(* IEC 61131-3 sources: elnaProjects/ElpcLogic/PomarKc7Changed/build_USO_ecl/_ (part 3) *)

  IF NOT onInit THEN
           fb_timer480(phaseNumber:=1, delay:=T#480S);
           fb_kran4Open(phaseNumber:=2, act:=_on);
           fb_waitAfterKran4(phaseNumber:=3, delay:=T#10S);
           fb_kran5Close(phaseNumber:=4, act:=_off);
           fb_kran3bOpen(phaseNumber:=5, act:=_on);
           fb_dP_kr1less100(phaseNumber:=6);
           fb_Pvh_vyhMore5(phaseNumber:=7);
           fb_kran1Open(phaseNumber:=8, act:=_on);
           fb_kran2Open(phaseNumber:=9, act:=_on);
           fb_kran3Open(phaseNumber:=10, act:=_on);
           fb_kran3bClose(phaseNumber:=11, act:=_off);
           fb_Err_ALG(phaseNumber:=12);
  onInit:=TRUE;
  END_IF;

  fb_timer480(StrPh:=timer480);
  fb_kran4Open(StrPh:= kran4Open, Im:=Im.kran4);
  fb_waitAfterKran4(StrPh:= waitAfterKran4);
  fb_kran5Close(StrPh:=kran5Close, Im:=Im.kran5);
  fb_kran3bOpen(StrPh:=kran3bOpen, Im:=Im.kran3b);
  fb_dP_kr1less100(StrPh:=dP_kr1less100);
  fb_Pvh_vyhMore5(StrPh:=Pvh_vyhMore5);
  fb_kran1Open(StrPh:=kran1Open, Im:=Im.kran1);
  fb_kran2Open(StrPh:=kran2Open, Im:=Im.kran2);
  fb_kran3Open(StrPh:=kran3Open, Im:=Im.kran3);
  fb_kran3bClose(StrPh:=kran3bClose, Im:=Im.kran3b);
  fb_Err_ALG(StrPh:=Err_ALG);

  StrAlg.CanRun := StrAlg.inCanRun;
  StrAlg.OpcCommandsDisabled := StrAlg.inOpcCommandsDisabled;

  IF StrAlg.isRuning THEN
      (* запуск таймера *)
      IF NOT (kran3bClose.top) THEN
  	    runPhase(timer480);
      END_IF;

      (*если кран1 не открыт - октрыть кран 4*)
      IF	NOT kran1Open.top (*AND IM.kran4._cmdreset.IN = FALSE*)  THEN
  	    runIfNotRunningSO(IM.SingleOutputs.Kr4_open_from_alg);
  	    runPhase(kran4Open);
      END_IF;
      IF	kran4Open.start AND NOT kran4Open.top THEN
  	    IF	IM.kran4.onStatus = _statusDualInput.STATUS_ON THEN
  		    kran4Open.top:=TRUE;
  	    END_IF;
      END_IF;

      (* продувка крана *)
      IF kran4Open.top THEN
          runPhase(waitAfterKran4);
      END_IF;

      (* кран продулся - закрытие кран 5*)
      IF waitAfterKran4.top THEN
  	    runPhase(kran5Close);
      END_IF;

      (* кран 5 закрыт - открытие крана 3б проверка перепада давление*)
      IF	kran5Close.top THEN
  	    runPhase(kran3bOpen);
  	    runPhase(dP_kr1less100);
  	    runPhase(Pvh_vyhMore5);
      END_IF;

      (* проверка давления крана *)
      IF	Pvh_vyhMore5.start AND NOT Pvh_vyhMore5.top THEN
  	    IF	(ai.Pgaza_na_vhode_nagnetatelia.interval >=statusAi.NORMAL) AND (ai.Pgaza_na_vhode_nagnetatelia.value	 >= 4.0) AND
  		    (ai.Pgaza_na_vyhode_nagnetatelia.interval >=statusAi.NORMAL) AND (ai.Pgaza_na_vyhode_nagnetatelia.value	 >= 4.0) THEN
  		        Pvh_vyhMore5.top := TRUE;
      		    runAiProtection(protections.Pgaza_na_vyhode_nagnetatelia);
  	    END_IF;
      END_IF;

      (* проверка открытия крана 3б *)
      IF	kran3bOpen.start AND NOT kran3bOpen.top THEN
  	    IF	IM.kran3b.onStatus=_statusDualInput.STATUS_ON THEN
  		    kran3bOpen.top :=TRUE;
  	    END_IF;
      END_IF;
      IF	kran3bOpen.top AND	kran5Close.top AND dP_kr1less100.top AND Pvh_vyhMore5.top THEN
  	    runPhase(kran1Open);
  	    runPhase(kran2Open);
  	    runPhase(kran3Open);
  	    (*Smazka_1_2:=TRUE; нет такого *)
      END_IF;
      IF	kran1Open.top THEN
  	    resetIfRunningSO(IM.SingleOutputs.Kr4_open_from_alg);
  	    (*ystavki.Block_kr4_alg.setValue (0);что такое уставки*)
      END_IF;

      (* закрытие крана 3бис *)
      IF kran1Open.top AND kran2Open.top AND kran3Open.top THEN
  	    runPhase(kran3bClose);
      END_IF;
      IF 	kran3bClose.top THEN
  	    Err_ALG.error :=FALSE;
  	    resetPhase(timer480);
      ELSIF NOT kran3bClose.top AND timer480.top THEN
  		Err_ALG.error :=TRUE;
      END_IF;
  END_IF;

  _sunpackerCommand(command := StrAlg.inCommand);
  	source := _sunpackerCommand.source;
  	cmd := _sunpackerCommand.cmd;

  IF cmd <> 0 AND lastCmd <> cmd AND (((NOT StrAlg.opcCommandsDisabled) AND source > 0) OR source = 0) then
  	CASE BYTE_TO_INT(cmd) OF
  		(*cmdRun*) 1: 	IF (StrAlg.CanRun) THEN
  					StrAlg.isRuning := TRUE;
  					StrAlg.isEnded := FALSE;
  					StrAlg.hasError := FALSE;
  					(*****************       OnRun       *****************)
                                                    algManager.nMode:=ModeGpa.MODE_PUSK_FIRST_FAZA2;

                                                    (*runPhase(timer120);
                                                    runPhase(timer5);
                                                    runPhase(Shup);
                                                    resetAiProtection(protections.dPmaslo_gaz);
                                                    resetDiProtection(protections.dPmaslo_gaz_less100);*)

  					cmd_for_Status := cmd;
  					source_for_Status := source;
  					command_error_for_Status := 0;
  				ELSE
  					StrAlg.isRuning := FALSE;
  					StrAlg.isEnded := FALSE;
  					StrAlg.hasError := FALSE;

  					cmd_for_Status := 0;
  					source_for_Status := source;
  					command_error_for_Status := cmd;
  				END_IF;
  		(*cmdReset*) 2: 	StrAlg.isRuning := FALSE;
  				StrAlg.isEnded := FALSE;
  				StrAlg.hasError 	:= FALSE;

                                           (*****************       OnReset       *****************)
                                          waitReset(IN:=FALSE);
                                          StrAlg.inCanRun:=FALSE;

                                          (*resetPhase(timer5);
                                          resetPhase(Shup);
                                          resetPhase(timer120);
                                          resetPhase(Net_Chast);
                                          resetPhase(mvOn);
                                          resetPhase(pGNSmore04);
                                          resetPhase(gotov_K_zagruzke);
                                          resetPhase(dPmg_Top);
                                          resetPhase(AutoPNS_Start);*)

                                          StrAlg.inOpcCommandsDisabled:=FALSE;

  				cmd_for_Status := cmd;
  				source_for_Status := source;
  				command_error_for_Status := 0;
  	END_CASE;
  	resetCmdTimer(IN := false);
  	resetCmdTimerPriznak := TRUE;
  END_IF;
  lastCmd := cmd;

  resetCmdTimer(IN := resetCmdTimerPriznak, PT := T#5S);
  IF resetCmdTimer.Q THEN
  	resetCmdTimerPriznak := FALSE;
  	source_for_Status := 0;
  	cmd_for_Status := 0;
  	command_error_for_Status := 0;
  END_IF;

  StrAlg.Start:= timer480.startStatus
              OR kran4Open.startStatus
              OR waitAfterKran4.startStatus
              OR kran5Close.startStatus
              OR kran3bOpen.startStatus
              OR dP_kr1less100.startStatus
              OR Pvh_vyhMore5.startStatus
              OR kran1Open.startStatus
              OR kran2Open.startStatus
              OR kran3Open.startStatus
              OR kran3bClose.startStatus
              OR Err_ALG.startStatus;

  StrAlg.Error := timer480.errorStatus
              OR kran4Open.errorStatus
              OR waitAfterKran4.errorStatus
              OR kran5Close.errorStatus
              OR kran3bOpen.errorStatus
              OR dP_kr1less100.errorStatus
              OR Pvh_vyhMore5.errorStatus
              OR kran1Open.errorStatus
              OR kran2Open.errorStatus
              OR kran3Open.errorStatus
              OR kran3bClose.errorStatus
              OR Err_ALG.errorStatus;

  StrAlg.Top := timer480.topStatus
              OR kran4Open.topStatus
              OR waitAfterKran4.topStatus
              OR kran5Close.topStatus
              OR kran3bOpen.topStatus
              OR dP_kr1less100.topStatus
              OR Pvh_vyhMore5.topStatus
              OR kran1Open.topStatus
              OR kran2Open.topStatus
              OR kran3Open.topStatus
              OR kran3bClose.topStatus
              OR Err_ALG.topStatus;

  (*TODO: TYPE PROGRAM CODE HERE*)
  StrAlg.status :=  SHL(BYTE_TO_DWORD(source_for_Status), 29)
  			OR SHL(BYTE_TO_DWORD(cmd_for_Status), 26)
  			OR SHL(BYTE_TO_DWORD(command_error_for_Status), 23)
  			OR SHL(BOOL_TO_DWORD(StrAlg.OpcCommandsDisabled ), 21)
  			OR SHL(BOOL_TO_DWORD(StrAlg.hasError),4)
  			OR SHL(BOOL_TO_DWORD(StrAlg.CanRun),2)
  			OR SHL(BOOL_TO_DWORD(StrAlg.isEnded),1)
  			OR BOOL_TO_DWORD(StrAlg.isRuning);
END_FUNCTION_BLOCK

FUNCTION_BLOCK fb_ph_SectionSwitch
  VAR_IN_OUT
    im : struct_SectionSwitch;
  END_VAR
  VAR_INPUT
    act : TYPE_DualStateImAction;
    PhaseNumber : UINT;
  END_VAR
  VAR_IN_OUT
    StrPh : struct_PhaseAlgoritm;
  END_VAR
  VAR
    CommandFault_Trig : R_TRIG;
    reset_Trig : R_TRIG;
    _statusDualInput : TYPE_statusDualInput;
  END_VAR

  IF StrPh.run AND NOT StrPh.start THEN
  	StrPh.start := TRUE;
  	StrPh.top := FALSE;
  	StrPh.error := FALSE;
            StrPh.run:=FALSE;

  	CASE act OF
  		(*DualStateImAction.on*)   _on : im.inOpcCommandsDisabled:=TRUE;
                                                       im.inCommand_Alg := 1; (*cmd_open*)
  		(*DualStateImAction.off*) _off : im.inOpcCommandsDisabled:=TRUE;
                                                       im.inCommand_Alg := 2; (*cmd_close*)
  	END_CASE;
  END_IF;

  IF StrPh.start AND NOT StrPh.top THEN
                      CommandFault_Trig(CLK := im.CommandFault);
                      IF CommandFault_Trig.Q THEN
  	          StrPh.error := TRUE;
                      END_IF;

  		CASE act OF
  		(*_DualStateImAction.on*)    _on: StrPh.top := im.onStatus = _statusDualInput.STATUS_ON;
  		(*_DualStateImAction.off*)  _off: StrPh.top := im.onStatus = _statusDualInput.STATUS_OFF;
  		END_CASE;

  END_IF;

  IF StrPh.top THEN
  StrPh.error := FALSE;
  END_IF;

  reset_Trig(CLK := StrPh.reset);
  IF reset_Trig.Q THEN
  	StrPh.start := FALSE;
  	StrPh.error := FALSE;
  	StrPh.top := FALSE;
            StrPh.run:=FALSE;
            StrPh.reset:=FALSE;
  END_IF;

  StrPh.startStatus := SHL(BOOL_TO_DWORD(StrPh.start), PhaseNumber);
  StrPh.errorStatus := SHL(BOOL_TO_DWORD(StrPh.error), PhaseNumber);
  StrPh.topStatus := SHL(BOOL_TO_DWORD(StrPh.top), PhaseNumber);
END_FUNCTION_BLOCK

FUNCTION_BLOCK Pusk_second_faza_reactor
  VAR_IN_OUT
    StrAlg : struct_Alg;
  END_VAR
  VAR
    timer25 : struct_PhaseAlgoritm;
    timer3 : struct_PhaseAlgoritm;
    mvOn : struct_PhaseAlgoritm;
    pGNSmore04 : struct_PhaseAlgoritm;
    gotov_K_zagruzke : struct_PhaseAlgoritm;
    dPmg_Top : struct_PhaseAlgoritm;
    Mv_Error : struct_PhaseAlgoritm;
    AutoPNS_Start : struct_PhaseAlgoritm;
    fb_timer25 : fb_ph_Timer;
    fb_timer3 : fb_ph_Timer;
    fb_Mv_Error : fb_ph_algoritm;
    fb_mvOn : fb_ph_SectionSwitch;
    fb_pGNSmore04 : fb_ph_algoritm;
    fb_gotov_K_zagruzke : fb_ph_algoritm;
    fb_dPmg_Top : fb_ph_algoritm;
    fb_AutoPNS_Start : fb_ph_algoritm;
    _sunpackerCommand : fb_sunpackerCommand;
    _statusDualInput : TYPE_statusDualInput;
    _Answers : TYPE_Answers;
    source : BYTE;
    cmd : BYTE;
    lastCmd : BYTE;
    source_for_Status : BYTE;
    cmd_for_Status : BYTE;
    command_error_for_Status : BYTE;
    resetCmdTimer : TON;
    resetCmdTimerPriznak : BOOL;
    onInit : BOOL;
    waitReset : TON;
  END_VAR
  VAR_EXTERNAL
    ModeGpa : TYPE_ModeGpa;
    algManager : struct_AlgoritmsManager;
    IM : ImConfig;
    protections : ProtectionsConfig;
    algoritms : AlgoritmsConfig;
    ai : AiConfig;
  END_VAR
  VAR
    statusAi : TYPE_StatusAi;
  END_VAR

  IF NOT onInit THEN
           fb_timer25(phaseNumber:=1, delay:=T#25S);
           fb_timer3(phaseNumber:=2, delay:=T#3S);
           fb_mvOn(phaseNumber:=3, act:=_on);
           fb_pGNSmore04(phaseNumber:=4);
           fb_gotov_K_zagruzke(phaseNumber:=5);
           fb_dPmg_Top(phaseNumber:=6);
           fb_Mv_Error(phaseNumber:=7);
           fb_AutoPNS_start(phaseNumber:=8, act:=_run, waitCompletion:=FALSE);

  onInit:=TRUE;
  END_IF;

  fb_timer25(StrPh:=timer25);
  fb_timer3(StrPh:= timer3);
  fb_mvOn(StrPh:= mvOn, Im:=IM.mv);
  fb_pGNSmore04(StrPh:=pGNSmore04);
  fb_gotov_K_zagruzke(StrPh:=gotov_K_zagruzke);
  fb_dPmg_Top(StrPh:=dPmg_Top);
  fb_Mv_Error(StrPh:=Mv_Error);
  fb_AutoPNS_start(StrPh:=AutoPNS_start, alg:=algoritms.autoPns);

  StrAlg.CanRun := StrAlg.inCanRun;
  StrAlg.OpcCommandsDisabled := StrAlg.inOpcCommandsDisabled;
  IF StrAlg.isRuning THEN
      (* если мв не завершен - включаем таймер *)
      IF NOT mvOn.top THEN
          runPhase(timer25);
      END_IF;

      (* если мв не заврешен - включаем таймер *)
      IF NOT mvOn.top THEN
          runPhase(timer3);
      END_IF;

      (* мв не запущен - запускаем мв *)
      IF NOT mvOn.start THEN
          runPhase(mvOn);
      END_IF;

      (* мв завершен *)
      IF mvOn.top  THEN
      (*если проверка пгнс не включена - включаем *)
          IF NOT pGNSmore04.start (*AND ((algManager.mode = modegpa.MODE_PUSKAP_R) OR (algManager.mode = modegpa.MODE_PUSKPP_R))*) THEN
              runPhase(pGNSmore04);
          END_IF;

          (*kakoito flag, hz zachem on
          IF NOT autoAVOM_canrun_flag THEN
              algoritms.S_AutoAVOM.CanRun:=TRUE;
              autoAVOM_canrun_flag:=TRUE;
          END_IF;*)
          resetPhase(timer3);
          resetPhase(timer25);
          Mv_Error.error := FALSE;
          runPhase(gotov_K_zagruzke);
          IF NOT dPmg_Top.start (*AND ((algManager.mode = modegpa.MODE_PUSKAP_R) OR (algManager.mode = modegpa.MODE_PUSKPP_R))*) THEN
              runPhase(dPmg_Top);
          END_IF;

          runDiProtection(protections.mvOff);
          runDiProtection(protections.Off_avar_vikluchatel);
          runDiProtection(protections.Reg_vozb_off);
          ELSIF NOT mvOn.top AND timer3.top THEN
  		Mv_Error.error := TRUE;
      END_IF;

      IF	dPmg_Top.start AND NOT dPmg_Top.top THEN
  	    IF	NOT IM.SingleSignals.dP_maslo_gaz_Less100.Q AND IM.SingleSignals.dP_maslo_gaz_Less100.status = 1 AND ai.dPmaslo_gaz.value > 150.0	THEN
  		    dPmg_Top.top:=TRUE;
  		    runAiProtection(protections.dPmaslo_gaz);
  		    runDiProtection(protections.dPmaslo_gaz_less100);
  		    resetAiProtection(protections.Pgaza_na_vhode_nagnetatelia_GPA_STOP);
  		    resetAiProtection(protections.Pgaza_na_vyhode_nagnetatelia_GPA_STOP);
  		    (*algoritms.autoNu_2.CanRun:=TRUE;
  		    algoritms.autoNu_2.run (); не понимаю*)
  	    END_IF;
      END_IF;

      IF	pGNSmore04.start AND NOT pGNSmore04.top THEN
  	    IF 	ai.Pmasla_posle_GNS.interval	>=statusAi.NORMAL AND ai.Pmasla_posle_GNS.value	 > 400.0 THEN
  	  	    pGNSmore04.top:=TRUE;
  	    END_IF;
      END_IF;

      IF	pGNSmore04.top AND gotov_K_zagruzke.top AND dPmg_Top.top (*AND algManager.mode = modegpa.MODE_PUSKAP_R) OR (algManager.mode = modegpa.MODE_PUSKPP_R)))*) OR
  	    gotov_K_zagruzke.top (*AND ((algManager.mode = modegpa.MODE_PUSKV_R) OR (algManager.mode = modegpa.MODE_I))))*) AND NOT AutoPNS_start.top  THEN
  	    algoritms.AutoPns.CanRun :=TRUE;
  	   (*algoritms.AutoPNS_Start.run();*)
  	    AutoPNS_start.top:=TRUE;
      END_IF;
      IF	timer25.top AND Mv_Error.error THEN
  	algoritms.ao.CanRun:=TRUE;
  	(*algoritms.ao.run ();*)
      END_IF;

      (*StrAlg.isEnded:= avom1cmdOff.top AND avom2cmdOff.top;*)
  END_IF;
  StrAlg.CanRun := StrAlg.inCanRun;
  StrAlg.OpcCommandsDisabled := StrAlg.inOpcCommandsDisabled;

  (* ---- Если управление с ВУ заблокировано, то  передаем команду из алгоритма ---- *)
  IF StrAlg.inOpcCommandsDisabled THEN
  	StrAlg.inCommand := StrAlg.inCommand_Alg;
  ELSE (* иначе передаем команду с АРМа*)
  	StrAlg.inCommand := StrAlg.inCommand_ARM;
  END_IF;

  _sunpackerCommand(command := StrAlg.inCommand);
  	source := _sunpackerCommand.source;
  	cmd := _sunpackerCommand.cmd;

  IF cmd <> 0 AND lastCmd <> cmd AND (((NOT StrAlg.opcCommandsDisabled) AND source > 0) OR source = 0) then
  	CASE BYTE_TO_INT(cmd) OF
  		(*cmdRun*) 1: 	IF (StrAlg.CanRun) THEN
  					StrAlg.isRuning := TRUE;
  					StrAlg.isEnded := FALSE;
  					StrAlg.hasError := FALSE;
  					(*****************       OnRun       *****************)
                                                    algManager.nMode:=ModeGpa.MODE_PUSK_FIRST_FAZA2;

                                                    (*runPhase(timer120);
                                                    runPhase(timer5);
                                                    runPhase(Shup);
                                                    resetAiProtection(protections.dPmaslo_gaz);
                                                    resetDiProtection(protections.dPmaslo_gaz_less100);*)

  					cmd_for_Status := cmd;
  					source_for_Status := source;
  					command_error_for_Status := 0;
  				ELSE
  					StrAlg.isRuning := FALSE;
  					StrAlg.isEnded := FALSE;
  					StrAlg.hasError := FALSE;

  					cmd_for_Status := 0;
  					source_for_Status := source;
  					command_error_for_Status := cmd;
  				END_IF;
  		(*cmdReset*) 2: 	StrAlg.isRuning := FALSE;
  				StrAlg.isEnded := FALSE;
  				StrAlg.hasError 	:= FALSE;

                                           (*****************       OnReset       *****************)
                                          waitReset(IN:=FALSE);
                                          StrAlg.inCanRun:=FALSE;

                                          (*resetPhase(timer5);
                                          resetPhase(Shup);
                                          resetPhase(timer120);
                                          resetPhase(Net_Chast);
                                          resetPhase(mvOn);
                                          resetPhase(pGNSmore04);
                                          resetPhase(gotov_K_zagruzke);
                                          resetPhase(dPmg_Top);
                                          resetPhase(AutoPNS_Start);*)

                                          StrAlg.inOpcCommandsDisabled:=FALSE;

  				cmd_for_Status := cmd;
  				source_for_Status := source;
  				command_error_for_Status := 0;
  	END_CASE;
  	resetCmdTimer(IN := false);
  	resetCmdTimerPriznak := TRUE;
  END_IF;
  lastCmd := cmd;

  resetCmdTimer(IN := resetCmdTimerPriznak, PT := T#5S);
  IF resetCmdTimer.Q THEN
  	resetCmdTimerPriznak := FALSE;
  	source_for_Status := 0;
  	cmd_for_Status := 0;
  	command_error_for_Status := 0;
  END_IF;

  StrAlg.Start:= timer25.errorStatus
              OR timer3.errorStatus
              OR mvOn.errorStatus
              OR pGNSmore04.errorStatus
              OR gotov_K_zagruzke.errorStatus
              OR dPmg_Top.errorStatus
              OR Mv_Error.errorStatus
              OR AutoPNS_Start.errorStatus;

  (*TODO: TYPE PROGRAM CODE HERE*)
  StrAlg.status :=  SHL(BYTE_TO_DWORD(source_for_Status), 29)
  			OR SHL(BYTE_TO_DWORD(cmd_for_Status), 26)
  			OR SHL(BYTE_TO_DWORD(command_error_for_Status), 23)
  			OR SHL(BOOL_TO_DWORD(StrAlg.OpcCommandsDisabled ), 21)
  			OR SHL(BOOL_TO_DWORD(StrAlg.hasError),4)
  			OR SHL(BOOL_TO_DWORD(StrAlg.CanRun),2)
  			OR SHL(BOOL_TO_DWORD(StrAlg.isEnded),1)
  			OR BOOL_TO_DWORD(StrAlg.isRuning);
END_FUNCTION_BLOCK

FUNCTION_BLOCK fb_KranOpenProtection
  VAR_INPUT
    im : struct_Kran;
  END_VAR
  VAR_IN_OUT
    StrDIp : struct_DiProtection;
  END_VAR
  VAR
    _sunpackerCommand : fb_sunpackerCommand;
    statusDualInput : TYPE_statusDualInput;
    _ProtectionTags : TYPE_ProtectionTags;
    _signalingTp : TOF;
    timer : TON;
    SignalingTrig : R_TRIG;
    SignalingFTrig : F_TRIG;
    SignalingDi : BOOL;
    source : BYTE;
    cmd : BYTE;
    lastCmd : BYTE;
    source_for_Status : BYTE;
    cmd_for_Status : BYTE;
    command_error_for_Status : BYTE;
    resetCmdTimer : TON;
    resetCmdTimerPriznak : BOOL;
    signalinTimer : TON;
    runOnStart_Trig : R_TRIG;
  END_VAR

  timer(IN := (im.onStatus<>statusDualInput.STATUS_ON) AND StrDIp.isRunning  , PT := StrDIp.delay);
  SignalingTrig(CLK := timer.Q);
  IF SignalingTrig.Q THEN
  	SignalingDi := TRUE;
  END_IF;
  SignalingFTrig(CLK := timer.Q);
  IF SignalingFTrig.Q THEN
  	SignalingDi := FALSE;
  END_IF;

  StrDIp.Tag := StrDIp.inTag;
  StrDIp.RunOnStart := StrDIp.inRunOnStart;

  StrDIp.CanRun := StrDIp.inCanRun;

  StrDIp.OpcCommandsDisabled := StrDIp.inOpcCommandsDisabled;

  (* ---- Если управление с ВУ заблокировано, то передаем команду из алгоритма ---- *)
  IF StrDIp.inOpcCommandsDisabled THEN
  	StrDIp.inCommand := StrDIp.inCommand_Alg;
  ELSE (* иначе передаем команду с АРМа*)
  	StrDIp.inCommand := StrDIp.inCommand_ARM;
  END_IF;

  _sunpackerCommand(command := StrDIp.inCommand);
  	source := _sunpackerCommand.source;
  	cmd := _sunpackerCommand.cmd;

  IF cmd <> 0 AND lastCmd <> cmd AND (((NOT StrDIp.opcCommandsDisabled) AND source > 0) OR source = 0) then
  	CASE BYTE_TO_INT(cmd) OF
  	        (*cmdRun*) 1: 	IF        NOT StrDIp.Remont THEN
  					StrDIp.isEnded := FALSE;
  					StrDIp.hasError 	:= FALSE;
  					StrDIp.isRunning := TRUE;
  					cmd_for_Status := cmd;
  					source_for_Status := source;
  					command_error_for_Status := 0;
  				ELSE
  					StrDIp.isRunning := FALSE;
  					StrDIp.isEnded := FALSE;
  					StrDIp.hasError 	:= FALSE;

  					cmd_for_Status := 0;
  					source_for_Status := source;
  					command_error_for_Status := cmd;
  				END_IF;
                                          StrDIp.inOpcCommandsDisabled:=FALSE;

                  (*cmdReset*) 2: 	StrDIp.isRunning := FALSE;
  				StrDIp.isEnded := FALSE;
  				StrDIp.hasError 	:= FALSE;
  				SignalingDi:= FALSE;
  				StrDIp.Check := FALSE;
  				cmd_for_Status := cmd;
  				source_for_Status := source;
  				command_error_for_Status := 0;
                                          StrDIp.inOpcCommandsDisabled:=FALSE;

  	(*cmd_setRemont*) 4 :	StrDIp.Remont := TRUE;
  				(*StrDIp.isRunning := FALSE;*)

  				cmd_for_Status := cmd;
  				source_for_Status := source;
  				command_error_for_Status := 0;

          (*cmd_resetRemont*) 5 : 	(*IF (im.onStatus<>statusDualInput.STATUS_ON) THEN
  					cmd_for_Status := 0;
  					source_for_Status := 0;
  					command_error_for_Status := cmd;
  				ELSE*)
  					StrDIp.Remont := FALSE;
  					(*StrDIp.isRunning := TRUE;*)

  					cmd_for_Status := cmd;
  					source_for_Status := source;
  					command_error_for_Status := 0;
  				(*END_IF;*)

  	(*cmd_setCheck*) 6 : 	StrDIp.Check := TRUE;

  				cmd_for_Status := cmd;
  				source_for_Status := source;
  				command_error_for_Status := 0;
  	END_CASE;
  	resetCmdTimer(IN := false);
  	resetCmdTimerPriznak := TRUE;
  END_IF;
  lastCmd := cmd;

  resetCmdTimer(IN := resetCmdTimerPriznak);
  IF resetCmdTimer.Q THEN
  	resetCmdTimerPriznak := FALSE;
  	source_for_Status := 0;
  	cmd_for_Status := 0;
  	command_error_for_Status := 0;
  END_IF;

  IF StrDIp.isRunning AND  NOT StrDIp.Remont AND NOT StrDIp.Check THEN
  	StrDIp.Signaling := SignalingDi;
  	StrDIp.SignalingTP := _signalingTp.Q;
  ELSE
  	StrDIp.Signaling := 0;
  	StrDIp.SignalingTP := 0;
  END_IF;

  _signalingTp(in := StrDIp.Signaling, PT := T#1s);

  StrDIp.status :=  SHL(BYTE_TO_DWORD(source_for_Status), 29)
  			OR SHL(BYTE_TO_DWORD(cmd_for_Status), 26)
  			OR SHL(BYTE_TO_DWORD(command_error_for_Status), 23)
  			OR SHL(BOOL_TO_DWORD(StrDIp.OpcCommandsDisabled ), 21)
  			OR SHL(BOOL_TO_DWORD(StrDIp.Signaling), 16)
  			OR SHL(BOOL_TO_DWORD(StrDIp.RunOnStart ), 15)
  			OR SHL(BOOL_TO_DWORD(StrDIp.remont), 6)
  			OR SHL(BOOL_TO_DWORD(StrDIp.Check), 5)
  			OR SHL(BOOL_TO_DWORD(StrDIp.hasError), 4)
  			OR SHL(BOOL_TO_DWORD(StrDIp.SignalingTP), 3)
  			OR SHL(BOOL_TO_DWORD(StrDIp.CanRun), 2)
  			OR SHL(BOOL_TO_DWORD(StrDIp.isEnded), 1)
  			OR BOOL_TO_DWORD(StrDIp.isRunning);
END_FUNCTION_BLOCK

FUNCTION_BLOCK fb_Kran
  VAR_INPUT
    statOn : BOOL;
    statOff : BOOL;
    statOn_reliability : BOOL;
    statOff_reliability : BOOL;
  END_VAR
  VAR_IN_OUT
    strKr : struct_Kran;
  END_VAR
  VAR_INPUT
    inNs : TYPE_ReliableBit;
    inAccident : TYPE_ReliableBit;
    inAuto : TYPE_ReliableBit;
    inManual : TYPE_ReliableBit;
    inLocal : TYPE_ReliableBit;
    inDistance : TYPE_ReliableBit;
    inErrorPowerOff : TYPE_ReliableBit;
    inErrorBlock : TYPE_ReliableBit;
    inSo : TYPE_ReliableBit;
    inSz : TYPE_ReliableBit;
    inDp : TYPE_ReliableBit;
  END_VAR
  VAR
    onInit : BOOL      := FALSE;
    _statOn : BOOL;
    _statOff : BOOL;
    getSdvig : BOOL;
    lastOnStatus : BYTE;
    cmd : BYTE;
    source : BYTE;
    lastCmd : BYTE;
    source_for_Status : BYTE;
    cmd_for_Status : BYTE;
    command_error_for_Status : BYTE;
    _sunpackerCommand : fb_sunpackerCommand;
    _statusDualInput : TYPE_statusDualInput;
    _commandDualInput : TYPE_commandDualInput;
    _commandErrorTimer : BOOL;
    resetErrorTimer : BOOL;
    _changWithoutCommand : BOOL;
    BlockedOpenControl : BOOL;
    errorCMDTimer : TON;
    _errorReset : TON;
    sdvigReset : TON;
    continueHoldCommandTimer : TON;
    outputsSets : TOF;
    dP_Trig : R_TRIG;
    dP_Trig_reliability : R_TRIG;
    resetBlockedOpenControl_Trig : R_TRIG;
  END_VAR
  VAR_IN_OUT
    cmdOn : BOOL;
    cmdOff : BOOL;
  END_VAR

  IF NOT onInit THEN
  IF strKr.ISVALIDREF_cmdOn XOR strKr.ISVALIDREF_cmdOff THEN
  	IF 	strKr.ISVALIDREF_cmdOn THEN
  		lastCmd:= 2; (*baseCmdOff*)
  	ELSE
  		lastCmd:= 1; (*baseCmdOn*)
  	END_IF;
  END_IF;
  onInit:=TRUE;
  END_IF;

  (* ---- Если управление с ВУ заблокировано, то в ИМ передаем команду из алгоритма ---- *)
  IF strKr.inOpcCommandsDisabled THEN
  	strKr.inCommand := strKr.inCommand_Alg;
  ELSE (* иначе передаем команду с АРМа*)
  	strKr.inCommand := strKr.inCommand_ARM;
  END_IF;

  (* ---- Формирование состояния механизма ---- *)

  IF (strKr.ISVALIDREF_statOn) OR (strKr.ISVALIDREF_statOff) THEN
  	IF (strKr.ISVALIDREF_statOn) AND (strKr.ISVALIDREF_statOff) THEN
  	strKr.reliability:= statOn_reliability AND statOff_reliability;
  		_statOn  := statOn;
  		_statOff := statOff;
  	ELSIF (strKr.ISVALIDREF_statOn) THEN
                       strKr.reliability:= statOn_reliability;
  		_statOn  := statOn;
  		_statOff := NOT statOn;
  	ELSIF (strKr.ISVALIDREF_statOff) THEN
  		 strKr.reliability:= statOff_reliability;
  		_statOn  := NOT statOff;
  		_statOff :=statOff;
  	END_IF;

  	IF strKr.reliability THEN
  		IF _statOn AND NOT _statOff 		THEN 	strKr.onStatus := _statusDualInput.STATUS_ON;
  		ELSIF _statOff AND NOT _statOn 	THEN 	strKr.onStatus := _statusDualInput.Status_OFF;
  		ELSIF NOT _statOn AND NOT _statOff 	THEN 	strKr.onStatus := _statusDualInput.STATUS_TRANSITIONAL;
  		ELSE					strKr.onStatus := _statusDualInput.STATUS_ERROR;
                      END_IF;

  	ELSE
  		strKr.onStatus := _statusDualInput.STATUS_NOTDEFINED;

  	END_IF;
  ELSE
  	CASE BYTE_TO_INT(lastCmd) OF
  		(*baseCmdOn*)  1: strKr.onStatus  := _statusDualInput.STATUS_ON;
  		(*baseCmdOff*) 2: strKr.onStatus  := _statusDualInput.STATUS_OFF;

  	ELSE
  		 strKr.onStatus := _statusDualInput.STATUS_NOTDEFINED;

  	END_CASE;
  END_IF;

  strKr.Accident := inAccident.value AND inAccident.reliability;
  strKr.Ns := inNs.value AND inNs.reliability;
  strKr.Auto := inAuto.value AND inAuto.reliability;
  strKr.Manual := inManual.value AND inManual.reliability;
  strKr.Local := inLocal.value AND inLocal.reliability;
  strKr.Distance := inDistance.value AND inDistance.reliability;
  strKr.ErrorPowerOff := inErrorPowerOff.value AND inErrorPowerOff.reliability;
  strKr.ErrorBlock := inErrorBlock.value AND inErrorBlock.reliability;
  strKr.OpcCommandsDisabled := strKr.inOpcCommandsDisabled;

  (* ---- Формирование признака блокировки Открытия крана по высокому давлению ---- *)
  	IF strKr.ISVALIDREF_inDp THEN

  		strKr.Dp := NOT inDp.value AND inDp.reliability;

  		dP_Trig(CLK := strKr.Dp );
  		dP_Trig_reliability(CLK :=NOT inDp.reliability);

  		IF dP_Trig.Q OR dP_Trig_reliability.Q THEN
  			BlockedOpenControl := TRUE;
  		END_IF;
  		(* ---- автоматический сброс *)
  		resetBlockedOpenControl_Trig(CLK := (inDp.value) AND inDp.reliability);
  		IF resetBlockedOpenControl_Trig.Q THEN
  			BlockedOpenControl := FALSE;
  		END_IF;
  	ELSE
  		strKr.Dp  := FALSE;
  		BlockedOpenControl := FALSE;
  	END_IF;

  (* ---- Формирование признака сдвига ---- *)
  getSdvig := FALSE;
  IF (strKr.ISVALIDREF_cmdOn OR strKr.ISVALIDREF_cmdOff) AND NOT strKr.Local THEN
  	IF NOT (strKr.CmdOn OR strKr.CmdOff) THEN
  		IF (lastOnStatus <> strKr.onStatus AND
  		(strKr.onStatus <> _statusDualInput.STATUS_NOTDEFINED AND strKr.onStatus <> _statusDualInput.STATUS_ERROR) AND
  		(lastOnStatus <> _statusDualInput.STATUS_NOTDEFINED AND lastOnStatus <> _statusDualInput.STATUS_ERROR)) THEN
  			strKr.sdvig   := TRUE;
  		END_IF;
  	END_IF;
  END_IF;

  IF getSdvig THEN strKr.sdvig:= TRUE; END_IF;

  sdvigReset(IN:=strKr.sdvig, PT:=T#15S);

  IF sdvigReset.Q THEN strKr.sdvig:=FALSE; END_IF;

  lastOnStatus := strKr.onStatus;

  (* ---- Распаковка команды ---- *)
  _sunpackerCommand(command := strKr.inCommand);
  	cmd := _sunpackerCommand.cmd;
  	source := _sunpackerCommand.source;

  (* ---- Обработка команды ---- *)
  IF cmd <> 0 AND lastCmd <> cmd and (((NOT strKr.opcCommandsDisabled) AND source > 0) OR source = 0) then
  	CASE BYTE_TO_INT(cmd) OF
  	(*cmd_open*) 1 :
  			IF NOT BlockedOpenControl THEN
                                IF  strKr.ISVALIDREF_cmdOn THEN strKr.CmdOn := TRUE;
  				IF strKr.ISVALIDREF_cmdOff THEN strKr.CmdOff := FALSE; END_IF;
  			ELSIF  strKr.ISVALIDREF_cmdOff THEN strKr.CmdOff := FALSE;  END_IF;
  			errorCMDTimer(IN := false);

  			_commandErrorTimer := true;
  			strKr.lastCmdIsOn := true;
                                END_IF;
  	(*cmd_close*) 2 :
  			IF strKr.ISVALIDREF_cmdOff THEN strKr.CmdOff := TRUE;
  				IF strKr.ISVALIDREF_cmdOn THEN strKr.CmdOn := FALSE; END_IF;
  			ELSIF strKr.ISVALIDREF_cmdOn THEN strKr.CmdOn := FALSE; END_IF;
  			errorCMDTimer(IN := false);

  			_commandErrorTimer := true;
  			strKr.lastCmdIsOn := false;
  	(*cmd_reset*) 3 :   IF (strKr.ISVALIDREF_statOn) OR (strKr.ISVALIDREF_statOff) THEN
  			strKr.CmdOn := FALSE;
  			strKr.CmdOff := FALSE;
                                lastCmd := 0;
  			_commandErrorTimer := false;
  			strKr.lastCmdIsOn := false;
                                END_IF;

  	END_CASE;
  	source_for_Status := source;
  	cmd_for_Status := cmd;
  	command_error_for_Status := 0;
  END_IF;
  lastCmd := cmd;

  errorCMDTimer(In := _commandErrorTimer, PT :=T#90s);

  continueHoldCommandTimer(IN:=(strKr.onStatus = _statusDualInput.STATUS_ON) OR
  (strKr.onStatus = _statusDualInput.STATUS_OFF), PT:=strKr.continueHoldCommand);

  (* ---- алгоритм  для команды ВКЛючить ---- *)
  IF (strKr.onStatus = _statusDualInput.STATUS_ON) and strKr.lastCmdIsOn  then
  	IF strKr.ISVALIDREF_cmdOn AND strKr.ISVALIDREF_cmdOff then
            IF continueHoldCommandTimer.Q THEN
            strKr.cmdOn := false; END_IF;
            END_IF;
  	 errorCMDTimer(In := false);
  	 _commandErrorTimer := false;
  	 cmd_for_Status := 0;
  	 source_for_Status := 0;
  END_IF;

  (* ---- off ---- *)
  IF (strKr.onStatus = _statusDualInput.STATUS_OFF) and  (NOT strKr.lastCmdIsOn) then
  	IF strKr.ISVALIDREF_cmdOn AND strKr.ISVALIDREF_cmdOff then
            IF continueHoldCommandTimer.Q THEN
            strKr.cmdOff := false; END_IF;
            END_IF;
  	 errorCMDTimer(In := false);
  	 _commandErrorTimer := false;
  	 cmd_for_Status := 0;
  	 source_for_Status := 0;
  END_IF;

  (* ---- ошибка исполнения команды ---- *)
  if errorCMDTimer.Q and (cmd_for_Status <> 0) then
  	command_error_for_Status :=  cmd_for_Status;
  	_commandErrorTimer := false;
  	strKr.CmdOn := false;
  	strKr.CmdOff := false;
  	(*lastCmd := 0;*)
  END_IF;

  (* ---- сброс ошибки команды ---- *)
  strKr.CommandFault := command_error_for_Status <> 0;
  _errorReset(IN := command_error_for_Status <> 0, PT := T#5S);
  IF _errorReset.Q THEN
  	cmd_for_Status := 0;
  	source_for_Status := 0;
  	command_error_for_Status := 0;

  END_IF;

  outputsSets(in := (strKr.ISVALIDREF_cmdOn and strKr.cmdOn ) OR (strKr.ISVALIDREF_cmdOff and strKr.cmdOff), PT := T#2S);
  	IF NOT outputsSets.Q THEN
  		strKr.So := inSo._inversed AND inSo.reliability AND strKr.ISVALIDREF_inSo;
  		strKr.Sz := inSz._inversed AND inSz.reliability AND strKr.ISVALIDREF_inSz;
  	END_IF;

  cmdOn := strKr.cmdOn;
  cmdOff:= strKr.cmdOff;

  (* ---- формирование зашифрованного статуса для АРМа ---- *)
  strKr.status := shl(BYTE_TO_DWORD(source_for_Status), 29)
  		OR shl(BYTE_TO_DWORD(cmd_for_Status), 26)
  		OR shl(BYTE_TO_DWORD(command_error_for_Status), 23)
  		OR shl(bool_to_DWORD(strKr.sdvig), 22)
  		OR shl(bool_to_DWORD(strKr.OpcCommandsDisabled), 21)
                      OR shl(bool_to_DWORD(strKr.Dp), 14)
                      OR shl(BOOL_TO_DWORD(strKr.Sz), 13)
  		OR shl(BOOL_TO_DWORD(strKr.So), 12)
  		OR shl(BOOL_TO_DWORD(strKr.ErrorBlock), 11)
  		OR shl(BOOL_TO_DWORD(strKr.ErrorPowerOff), 10)
  		OR shl(BOOL_TO_DWORD(strKr.Manual), 8)
  		OR shl(BOOL_TO_DWORD(strKr.Auto), 7)
  		OR shl(BOOL_TO_DWORD(strKr.Distance), 6)
  		OR shl(BOOL_TO_DWORD(strKr.Local), 5)
  		OR shl(BOOL_TO_DWORD(strKr.Ns), 4)
                  	OR shl(BOOL_TO_DWORD(strKr.Accident ),3)
  		OR BYTE_TO_DWORD(strKr.onStatus);
END_FUNCTION_BLOCK

FUNCTION_BLOCK fb_TableValue_Min
  VAR_INPUT
    parametr : REAL;
  END_VAR
  VAR
    _table : ARRAY [0..8] OF TYPE_TableRec;
  END_VAR
  VAR_INPUT
    inverse : BOOL      := FALSE;
  END_VAR
  VAR_IN_OUT
    actualValue : REAL;
  END_VAR
  VAR
    indexLess : INT      := -1;
    indexMore : INT      := -1;
    Vali : REAL;
    i : INT;
    moreDistance : REAL;
    lessDistance : REAL;
    onInit : BOOL;
    _prevParam : REAL      := 50.0;
  END_VAR
  VAR CONSTANT
    maxTableLength : INT      := 9;
  END_VAR

  IF NOT onInit THEN
  _table[0].x:=-35.0;  _table[0].y:=130.0;
  _table[1].x:=-25.0;  _table[1].y:=124.0;
  _table[2].x:=-15.0;  _table[2].y:=118.0;
  _table[3].x:= -5.0;  _table[3].y:=112.0;
  _table[4].x:=  0.0;  _table[4].y:=108.0;
  _table[5].x:=  5.0;  _table[5].y:=106.0;
  _table[6].x:= 15.0;  _table[6].y:=104.0;
  _table[7].x:= 25.0;  _table[7].y:=102.0;
  _table[8].x:= 35.0;  _table[8].y:= 97.0;

  onInit:=TRUE;
  END_IF;

  IF parametr <> _prevParam THEN
  indexLess:=-1;
  indexMore:=-1;
  lessDistance:=0.0;
  moreDistance:=0.0;
  FOR i:=0 TO maxTableLength-1 DO
  	IF NOT inverse THEN
  		Vali:=_table[i].x;
  	ELSE
  		Vali:=_table[i].y;
  	END_IF;

  	IF (Vali=parametr) THEN
  		indexLess:=i;
  		indexMore:=i;
  	ELSIF ((Vali<parametr) AND ((lessDistance>parametr-Vali) OR (indexLess<0))) THEN
  		indexLess:=i;
  		lessDistance:=parametr-Vali;
  	ELSIF ((Vali>parametr) AND ((moreDistance>Vali-parametr) OR (indexMore<0))) THEN
  		indexMore:=i;
  		moreDistance:=parametr-Vali;
  	END_IF;
  END_FOR;
  (*
  IF indexLess<0 THEN
  	indexLess:=indexMore;
  END_IF;

  IF indexMore<0 THEN
  	indexMore:=indexLess;
  END_IF;
  *)
    IF (_table[indexMore].x<>_table[indexLess].x) THEN
    actualValue:=_table[indexLess].y+((_table[indexMore].y-_table[indexLess].y)/(_table[indexMore].x-_table[indexLess].x))*(parametr-_table[indexLess].x);
    ELSE
    actualValue:=_table[indexLess].y;
    END_IF;
     _prevParam:= parametr;
  END_IF;
END_FUNCTION_BLOCK

FUNCTION_BLOCK fb_TableValue_Max
  VAR_INPUT
    parametr : REAL;
  END_VAR
  VAR
    _table : ARRAY [0..8] OF TYPE_TableRec;
  END_VAR
  VAR_INPUT
    inverse : BOOL      := FALSE;
  END_VAR
  VAR_IN_OUT
    actualValue : REAL;
  END_VAR
  VAR
    indexLess : INT      := -1;
    indexMore : INT      := -1;
    Vali : REAL;
    i : INT;
    moreDistance : REAL;
    lessDistance : REAL;
    onInit : BOOL;
    _prevParam : REAL      := 50.0;
  END_VAR
  VAR CONSTANT
    maxTableLength : INT      := 9;
  END_VAR

  IF NOT onInit THEN
  _table[0].x:=-35.0;  _table[0].y:=320.0;
  _table[1].x:=-25.0;  _table[1].y:=315.0;
  _table[2].x:=-15.0;  _table[2].y:=310.0;
  _table[3].x:= -5.0;  _table[3].y:=305.0;
  _table[4].x:=  0.0;  _table[4].y:=300.0;
  _table[5].x:=  5.0;  _table[5].y:=295.0;
  _table[6].x:= 15.0;  _table[6].y:=290.0;
  _table[7].x:= 25.0;  _table[7].y:=285.0;
  _table[8].x:= 35.0;  _table[8].y:=280.0;

  onInit:=TRUE;
  END_IF;

  IF parametr <> _prevParam THEN
  indexLess:=-1;
  indexMore:=-1;
  lessDistance:=0.0;
  moreDistance:=0.0;
  FOR i:=0 TO maxTableLength-1 DO
  	IF NOT inverse THEN
  		Vali:=_table[i].x;
  	ELSE
  		Vali:=_table[i].y;
  	END_IF;

  	IF (Vali=parametr) THEN
  		indexLess:=i;
  		indexMore:=i;
  	ELSIF ((Vali<parametr) AND ((lessDistance>parametr-Vali) OR (indexLess<0))) THEN
  		indexLess:=i;
  		lessDistance:=parametr-Vali;
  	ELSIF ((Vali>parametr) AND ((moreDistance>Vali-parametr) OR (indexMore<0))) THEN
  		indexMore:=i;
  		moreDistance:=parametr-Vali;
  	END_IF;
  END_FOR;
  (*
  IF indexLess<0 THEN
  	indexLess:=indexMore;
  END_IF;

  IF indexMore<0 THEN
  	indexMore:=indexLess;
  END_IF;
  *)
    IF (_table[indexMore].x<>_table[indexLess].x) THEN
    actualValue:=_table[indexLess].y+((_table[indexMore].y-_table[indexLess].y)/(_table[indexMore].x-_table[indexLess].x))*(parametr-_table[indexLess].x);
    ELSE
    actualValue:=_table[indexLess].y;
    END_IF;
     _prevParam:= parametr;
  END_IF;
END_FUNCTION_BLOCK

FUNCTION_BLOCK fb_RashodAlg
  VAR_INPUT
    P_gasIn : struct_AI;
  END_VAR
  VAR_IN_OUT
    StrAi : struct_AI;
  END_VAR
  VAR_INPUT
    T_gasIn : struct_AI;
    dP_konf : struct_AI;
    K : struct_AnalogParametr;
    A : struct_AnalogParametr;
    y0 : struct_AnalogParametr;
  END_VAR
  VAR
    num : LREAL;
    den : LREAL;
    _statusAi : TYPE_StatusAi;
  END_VAR
  VAR CONSTANT
    P0 : LREAL      := 0.1033;
    T0 : LREAL      := 293.0;
  END_VAR

  strAI.opcCommandsDisabled := strAI.inopcCommandsDisabled ;

  IF (P_gasIn.interval < _statusAi.normal) OR
     (T_gasIn.interval < _statusAi.normal) OR
     (dP_konf.interval < _statusAi.normal) THEN
  	StrAi.interval := _statusAi.NOTRELIABLE;
            strAI.status := 	SHL(BOOL_TO_DWORD(strAI.OpcCommandsDisabled ), 21)
  	OR BYTE_TO_DWORD(strAI.interval);
  	RETURN;
  END_IF;

  IF (P_gasIn.value <0.3) THEN
  	StrAi.interval := _statusAi.normal;
  	StrAi.value:= 0.0;
            strAI.status := 	SHL(BOOL_TO_DWORD(strAI.OpcCommandsDisabled ), 21)
  	OR BYTE_TO_DWORD(strAI.interval);
  	RETURN;
  END_IF;

  StrAi.interval:= _statusAi.normal;

  num:= (dP_konf.Value/1000.0)*(T_gasIn.value+273.0)*P0*735.56*K.Value;
  den:= y0.Value*P_gasIn.value*T0 ;

  StrAi.value:= A.Value*SQRT(num/den);

  strAI.status := 	SHL(BOOL_TO_DWORD(strAI.OpcCommandsDisabled ), 21) (* Управление в ВУ заблокировано *)
  		OR BYTE_TO_DWORD(strAI.interval);	              (* интервал *)
END_FUNCTION_BLOCK

FUNCTION_BLOCK fb_ZapasAlg
  VAR_INPUT
    Q_actual : struct_AI;
  END_VAR
  VAR_IN_OUT
    StrAi : struct_AI;
  END_VAR
  VAR_INPUT
    Q_min : LREAL;
    Q_max : LREAL;
  END_VAR
  VAR
    _statusAi : TYPE_StatusAi;
  END_VAR

  IF (Q_actual.interval < _statusAi.normal) THEN
  	StrAi.interval := _statusAi.NOTRELIABLE;
            strAI.status := 	SHL(BOOL_TO_DWORD(strAI.OpcCommandsDisabled ), 21)
  		OR BYTE_TO_DWORD(strAI.interval);
  	RETURN;
  END_IF;

  IF (Q_actual.value <10.0) THEN
  	StrAi.interval := _statusAi.normal;
  	StrAi.value:= 100.0;
            strAI.status := 	SHL(BOOL_TO_DWORD(strAI.OpcCommandsDisabled ), 21)
  		OR BYTE_TO_DWORD(strAI.interval);
  	RETURN;
  END_IF;

  strAI.opcCommandsDisabled := strAI.inopcCommandsDisabled ;
  StrAi.interval:= _statusAi.normal;

  StrAi.value:= ((Q_actual.value - Q_min)/(Q_max-Q_min))*100.0;

  strAI.status := 	SHL(BOOL_TO_DWORD(strAI.OpcCommandsDisabled ), 21) (* Управление в ВУ заблокировано *)
  		OR BYTE_TO_DWORD(strAI.interval);	              (* интервал *)
END_FUNCTION_BLOCK

FUNCTION_BLOCK fb_AntiPompagAlg
  VAR
    tableQ_min : fb_TableValue_Min;
    tableQ_max : fb_TableValue_Max;
    fb_Rashod : fb_RashodAlg;
    fb_Zapas : fb_ZapasAlg;
  END_VAR
  VAR_IN_OUT
    Kran6 : struct_Kran;
    StrAlg : struct_Alg;
    Rashod : struct_AI;
    Zapas : struct_AI;
  END_VAR
  VAR_INPUT
    P_gasIn : struct_AI;
    T_gasIn : struct_AI;
    dP_konf : struct_AI;
    UgolVNA : struct_AnalogParametr;
    K : struct_AnalogParametr;
    A : struct_AnalogParametr;
    y0 : struct_AnalogParametr;
  END_VAR
  VAR
    Q_max : LREAL;
    Q_min : LREAL;
    pompaj : BOOL;
    _statusAi : TYPE_StatusAi;
    _statusDualInput : TYPE_statusDualInput;
    _sunpackerCommand : fb_sunpackerCommand;
    source : BYTE;
    cmd : BYTE;
    lastCmd : BYTE;
    source_for_Status : BYTE;
    cmd_for_Status : BYTE;
    command_error_for_Status : BYTE;
    resetCmdTimer : TON;
    resetCmdTimerPriznak : BOOL;
  END_VAR

  tableQ_min(parametr:=LREAL_TO_REAL(UgolVNA.Value));

  tableQ_max(parametr:=LREAL_TO_REAL(UgolVNA.Value));

  Q_min:=REAL_TO_LREAL(tableQ_min.actualValue);

  Q_max:=REAL_TO_LREAL(tableQ_max.actualValue);

  fb_Rashod(StrAi:=Rashod, P_gasIn:=P_gasIn, T_gasIn:=T_gasIn, dP_konf:=dP_konf, K:=K, A:=A, y0:=y0);

  fb_Zapas(StrAi:=Zapas, Q_actual:=Rashod, Q_min:=Q_min, Q_max:=Q_max);

  StrAlg.CanRun := StrAlg.inCanRun;

  StrAlg.OpcCommandsDisabled := StrAlg.inOpcCommandsDisabled;

  IF StrAlg.isRuning THEN

  StrAlg.hasError := (Rashod.interval < _statusAi.normal);

  pompaj:= (Rashod.interval>=_statusAi.normal) AND (Rashod.value <= Q_min);

  IF pompaj THEN
            Kran6.inOpcCommandsDisabled:=TRUE;
  	Kran6.inCommand_Alg := 1;  (*cmd_open*)
  END_IF;

  StrAlg.isEnded := Kran6.onStatus = _statusDualInput.STATUS_ON ;

  END_IF;

  (* ---- Если управление с ВУ заблокировано, то передаем команду из алгоритма ---- *)
  IF StrAlg.inOpcCommandsDisabled THEN
  	StrAlg.inCommand := StrAlg.inCommand_Alg;
  ELSE (* иначе передаем команду с АРМа*)
  	StrAlg.inCommand := StrAlg.inCommand_ARM;
  END_IF;

  _sunpackerCommand(command := StrAlg.inCommand);
  	source := _sunpackerCommand.source;
  	cmd := _sunpackerCommand.cmd;

  IF cmd <> 0 AND lastCmd <> cmd AND (((NOT StrAlg.opcCommandsDisabled) AND source > 0) OR source = 0) then
  	CASE BYTE_TO_INT(cmd) OF
  		(*cmdRun*) 1: 	IF (StrAlg.CanRun) THEN
  					StrAlg.isRuning := TRUE;
  					StrAlg.isEnded := FALSE;
  					StrAlg.hasError 	:= FALSE;

                                                    (*****************       OnRun       *****************)

  					cmd_for_Status := cmd;
  					source_for_Status := source;
  					command_error_for_Status := 0;
  				ELSE
  					StrAlg.isRuning := FALSE;
  					StrAlg.isEnded := FALSE;
  					StrAlg.hasError 	:= FALSE;

  					cmd_for_Status := 0;
  					source_for_Status := source;
  					command_error_for_Status := cmd;
  				END_IF;
  		(*cmdReset*) 2: 	StrAlg.isRuning := FALSE;
  				StrAlg.isEnded := FALSE;
  				StrAlg.hasError 	:= FALSE;
                                          (*****************       OnReset       *****************)

                                                    pompaj:= FALSE;
                                                    Kran6.inOpcCommandsDisabled:=FALSE;
  				cmd_for_Status := cmd;
  				source_for_Status := source;
  				command_error_for_Status := 0;
  	END_CASE;
  	resetCmdTimer(IN := false);
  	resetCmdTimerPriznak := TRUE;
  END_IF;
  lastCmd := cmd;

  resetCmdTimer(IN := resetCmdTimerPriznak, PT := T#5S);
  IF resetCmdTimer.Q THEN
  	resetCmdTimerPriznak := FALSE;
  	source_for_Status := 0;
  	cmd_for_Status := 0;
  	command_error_for_Status := 0;
  END_IF;

  StrAlg.status :=  SHL(BYTE_TO_DWORD(source_for_Status), 29)
  			OR SHL(BYTE_TO_DWORD(cmd_for_Status), 26)
  			OR SHL(BYTE_TO_DWORD(command_error_for_Status), 23)
  			OR SHL(BOOL_TO_DWORD(StrAlg.OpcCommandsDisabled ), 21)
  			OR SHL(BOOL_TO_DWORD(StrAlg.hasError),4)
  			OR SHL(BOOL_TO_DWORD(StrAlg.CanRun),2)
  			OR SHL(BOOL_TO_DWORD(StrAlg.isEnded),1)
  			OR BOOL_TO_DWORD(StrAlg.isRuning);
END_FUNCTION_BLOCK

FUNCTION_BLOCK fb_AnalogParametr_Init
  VAR_INPUT
    data_Ini : BOOL;
    currentValue : LREAL;
    minVal : LREAL;
    maxVal : LREAL;
    maxStep : LREAL;
    minVal_ISVALIDREF : BOOL;
    maxVal_ISVALIDREF : BOOL;
    maxStep_ISVALIDREF : BOOL;
  END_VAR
  VAR_IN_OUT
    strAP : struct_AnalogParametr;
  END_VAR
  VAR_OUTPUT
    Init : BOOL      := FALSE;
  END_VAR

  (*****            Функциональный блок переинициализации Аналогового параметра.            *****)
       Init := false;

      IF data_Ini THEN                            (* Параметрам требуется переинициализация. *)
          strAP.currentValue          := currentValue;
          strAP.minVal                := minVal;
          strAP.maxVal                := maxVal;
          strAP.maxStep               := maxStep;
          strAP.minVal_ISVALIDREF     := minVal_ISVALIDREF;
          strAP.maxVal_ISVALIDREF     := maxVal_ISVALIDREF;
          strAP.maxStep_ISVALIDREF    := maxStep_ISVALIDREF;

          data_Ini:=false;
          Init := TRUE;
       END_IF;
       IF Init THEN
          currentValue:= 0.0;
          minVal:= 0.0;
          maxVal:= 0.0;
          maxStep:= 0.0;
          minVal_ISVALIDREF:= false;
          maxVal_ISVALIDREF:= false;
          maxStep_ISVALIDREF:= false;
       END_IF;
END_FUNCTION_BLOCK

FUNCTION_BLOCK fb_MvProtection
  VAR_INPUT
    sw : struct_SectionSwitch;
  END_VAR
  VAR_IN_OUT
    StrDIp : struct_DiProtection;
  END_VAR
  VAR
    _sunpackerCommand : fb_sunpackerCommand;
    statusDualInput : TYPE_statusDualInput;
    _ProtectionTags : TYPE_ProtectionTags;
    _signalingTp : TOF;
    timer : TON;
    SignalingTrig : R_TRIG;
    SignalingFTrig : F_TRIG;
    SignalingDi : BOOL;
    source : BYTE;
    cmd : BYTE;
    lastCmd : BYTE;
    source_for_Status : BYTE;
    cmd_for_Status : BYTE;
    command_error_for_Status : BYTE;
    resetCmdTimer : TON;
    resetCmdTimerPriznak : BOOL;
    signalinTimer : TON;
    runOnStart_Trig : R_TRIG;
  END_VAR

  timer(IN := (sw.onStatus = statusDualInput.STATUS_OFF) AND StrDIp.isRunning  , PT := StrDIp.delay);
  SignalingTrig(CLK := timer.Q);
  IF SignalingTrig.Q THEN
  	SignalingDi := TRUE;
  END_IF;
  SignalingFTrig(CLK := timer.Q);
  IF SignalingFTrig.Q THEN
  	SignalingDi := FALSE;
  END_IF;

  StrDIp.Tag := StrDIp.inTag;
  StrDIp.RunOnStart := StrDIp.inRunOnStart;

  StrDIp.CanRun := StrDIp.inCanRun;

  StrDIp.OpcCommandsDisabled := StrDIp.inOpcCommandsDisabled;

  (* ---- Если управление с ВУ заблокировано, то передаем команду из алгоритма ---- *)
  IF StrDIp.inOpcCommandsDisabled THEN
  	StrDIp.inCommand := StrDIp.inCommand_Alg;
  ELSE (* иначе передаем команду с АРМа*)
  	StrDIp.inCommand := StrDIp.inCommand_ARM;
  END_IF;

  _sunpackerCommand(command := StrDIp.inCommand);
  	source := _sunpackerCommand.source;
  	cmd := _sunpackerCommand.cmd;

  IF cmd <> 0 AND lastCmd <> cmd AND (((NOT StrDIp.opcCommandsDisabled) AND source > 0) OR source = 0) then
  	CASE BYTE_TO_INT(cmd) OF
  	        (*cmdRun*) 1: 	IF        NOT StrDIp.Remont THEN
  					StrDIp.isEnded := FALSE;
  					StrDIp.hasError 	:= FALSE;
  					StrDIp.isRunning := TRUE;
  					cmd_for_Status := cmd;
  					source_for_Status := source;
  					command_error_for_Status := 0;
  				ELSE
  					StrDIp.isRunning := FALSE;
  					StrDIp.isEnded := FALSE;
  					StrDIp.hasError 	:= FALSE;

  					cmd_for_Status := 0;
  					source_for_Status := source;
  					command_error_for_Status := cmd;
  				END_IF;
                                          StrDIp.inOpcCommandsDisabled:=FALSE;

                  (*cmdReset*) 2: 	StrDIp.isRunning := FALSE;
  				StrDIp.isEnded := FALSE;
  				StrDIp.hasError 	:= FALSE;
  				SignalingDi:= FALSE;
  				StrDIp.Check := FALSE;
  				cmd_for_Status := cmd;
  				source_for_Status := source;
  				command_error_for_Status := 0;
                                          StrDIp.inOpcCommandsDisabled:=FALSE;

  	(*cmd_setRemont*) 4 :	StrDIp.Remont := TRUE;
  				(*StrDIp.isRunning := FALSE;*)

  				cmd_for_Status := cmd;
  				source_for_Status := source;
  				command_error_for_Status := 0;

          (*cmd_resetRemont*) 5 : 	(*IF (sw.onStatus = statusDualInput.STATUS_OFF) THEN
  					cmd_for_Status := 0;
  					source_for_Status := 0;
  					command_error_for_Status := cmd;
  				ELSE*)
  					StrDIp.Remont := FALSE;
  					(*StrDIp.isRunning := TRUE;*)

  					cmd_for_Status := cmd;
  					source_for_Status := source;
  					command_error_for_Status := 0;
  				(*END_IF;*)

  	(*cmd_setCheck*) 6 : 	StrDIp.Check := TRUE;

  				cmd_for_Status := cmd;
  				source_for_Status := source;
  				command_error_for_Status := 0;
  	END_CASE;
  	resetCmdTimer(IN := false);
  	resetCmdTimerPriznak := TRUE;
  END_IF;
  lastCmd := cmd;

  resetCmdTimer(IN := resetCmdTimerPriznak);
  IF resetCmdTimer.Q THEN
  	resetCmdTimerPriznak := FALSE;
  	source_for_Status := 0;
  	cmd_for_Status := 0;
  	command_error_for_Status := 0;
  END_IF;

  IF StrDIp.isRunning AND  NOT StrDIp.Remont AND NOT StrDIp.Check THEN
  	StrDIp.Signaling := SignalingDi;
  	StrDIp.SignalingTP := _signalingTp.Q;
  ELSE
  	StrDIp.Signaling := 0;
  	StrDIp.SignalingTP := 0;
  END_IF;

  _signalingTp(in := StrDIp.Signaling, PT := T#1s);

  StrDIp.status :=  SHL(BYTE_TO_DWORD(source_for_Status), 29)
  			OR SHL(BYTE_TO_DWORD(cmd_for_Status), 26)
  			OR SHL(BYTE_TO_DWORD(command_error_for_Status), 23)
  			OR SHL(BOOL_TO_DWORD(StrDIp.OpcCommandsDisabled ), 21)
  			OR SHL(BOOL_TO_DWORD(StrDIp.Signaling), 16)
  			OR SHL(BOOL_TO_DWORD(StrDIp.RunOnStart ), 15)
  			OR SHL(BOOL_TO_DWORD(StrDIp.remont), 6)
  			OR SHL(BOOL_TO_DWORD(StrDIp.Check), 5)
  			OR SHL(BOOL_TO_DWORD(StrDIp.hasError), 4)
  			OR SHL(BOOL_TO_DWORD(StrDIp.SignalingTP), 3)
  			OR SHL(BOOL_TO_DWORD(StrDIp.CanRun), 2)
  			OR SHL(BOOL_TO_DWORD(StrDIp.isEnded), 1)
  			OR BOOL_TO_DWORD(StrDIp.isRunning);
END_FUNCTION_BLOCK

FUNCTION_BLOCK fb_DiProtection
  VAR_INPUT
    di : struct_singleSignal;
  END_VAR
  VAR_IN_OUT
    StrDIp : struct_DiProtection;
  END_VAR
  VAR
    _sunpackerCommand : fb_sunpackerCommand;
    _ProtectionTags : TYPE_ProtectionTags;
    _signalingTp : TOF;
    timer : TON;
    SignalingTrig : R_TRIG;
    SignalingFTrig : F_TRIG;
    SignalingDi : BOOL;
    source : BYTE;
    cmd : BYTE;
    lastCmd : BYTE;
    source_for_Status : BYTE;
    cmd_for_Status : BYTE;
    command_error_for_Status : BYTE;
    resetCmdTimer : TON;
    resetCmdTimerPriznak : BOOL;
    signalinTimer : TON;
    runOnStart_Trig : R_TRIG;
  END_VAR

  timer(IN := di.Q AND StrDIp.isRunning  , PT := StrDIp.delay);
  SignalingTrig(CLK := timer.Q);
  IF SignalingTrig.Q THEN
  	SignalingDi := TRUE;
  END_IF;
  SignalingFTrig(CLK := timer.Q);
  IF SignalingFTrig.Q THEN
  	SignalingDi := FALSE;
  END_IF;

  StrDIp.Tag := StrDIp.inTag;
  StrDIp.RunOnStart := StrDIp.inRunOnStart;

  StrDIp.CanRun := StrDIp.inCanRun;

  StrDIp.OpcCommandsDisabled := StrDIp.inOpcCommandsDisabled;

  (* ---- Если управление с ВУ заблокировано, то передаем команду из алгоритма ---- *)
  IF StrDIp.inOpcCommandsDisabled THEN
  	StrDIp.inCommand := StrDIp.inCommand_Alg;
  ELSE (* иначе передаем команду с АРМа*)
  	StrDIp.inCommand := StrDIp.inCommand_ARM;
  END_IF;

  _sunpackerCommand(command := StrDIp.inCommand);
  	source := _sunpackerCommand.source;
  	cmd := _sunpackerCommand.cmd;

  IF cmd <> 0 AND lastCmd <> cmd AND (((NOT StrDIp.opcCommandsDisabled) AND source > 0) OR source = 0) then

  	CASE BYTE_TO_INT(cmd) OF
  	        (*cmdRun*) 1: 	IF        NOT StrDIp.Remont THEN
  					StrDIp.isEnded := FALSE;
  					StrDIp.hasError 	:= FALSE;
  					StrDIp.isRunning := TRUE;
  					cmd_for_Status := cmd;
  					source_for_Status := source;
  					command_error_for_Status := 0;
  				ELSE
  					StrDIp.isRunning := FALSE;
  					StrDIp.isEnded := FALSE;
  					StrDIp.hasError 	:= FALSE;

  					cmd_for_Status := 0;
  					source_for_Status := source;
  					command_error_for_Status := cmd;
  				END_IF;
                                          StrDIp.inOpcCommandsDisabled:=FALSE;

                  (*cmdReset*) 2: 	StrDIp.isRunning := FALSE;
  				StrDIp.isEnded := FALSE;
  				StrDIp.hasError 	:= FALSE;
  				SignalingDi:= FALSE;
  				StrDIp.Check := FALSE;
  				cmd_for_Status := cmd;
  				source_for_Status := source;
  				command_error_for_Status := 0;
                                         StrDIp.inOpcCommandsDisabled:=FALSE;

  	(*cmd_setRemont*) 4 :	StrDIp.Remont := TRUE;
  				(*StrDIp.isRunning := FALSE;*)

  				cmd_for_Status := cmd;
  				source_for_Status := source;
  				command_error_for_Status := 0;
          (*cmd_resetRemont*) 5 : 	(*IF di.Q THEN
  					cmd_for_Status := 0;
  					source_for_Status := 0;
  					command_error_for_Status := cmd;
  				ELSE*)
  					StrDIp.Remont := FALSE;
  					(*StrDIp.isRunning := TRUE;*)

  					cmd_for_Status := cmd;
  					source_for_Status := source;
  					command_error_for_Status := 0;
  				(*END_IF;*)
  	(*cmd_setCheck*) 6 : 	StrDIp.Check := TRUE;

  				cmd_for_Status := cmd;
  				source_for_Status := source;
  				command_error_for_Status := 0;
  	END_CASE;
  	resetCmdTimer(IN := false);
  	resetCmdTimerPriznak := TRUE;
  END_IF;
  lastCmd := cmd;

  resetCmdTimer(IN := resetCmdTimerPriznak);
  IF resetCmdTimer.Q THEN
  	resetCmdTimerPriznak := FALSE;
  	source_for_Status := 0;
  	cmd_for_Status := 0;
  	command_error_for_Status := 0;
  END_IF;

  IF StrDIp.isRunning AND NOT StrDIp.Remont AND NOT StrDIp.Check THEN
  	StrDIp.Signaling := SignalingDi;
  	StrDIp.SignalingTP := _signalingTp.Q;
  ELSE
  	StrDIp.Signaling := 0;
  	StrDIp.SignalingTP := 0;
  END_IF;

  _signalingTp(in := StrDIp.Signaling, PT := T#1s);

  StrDIp.status :=  SHL(BYTE_TO_DWORD(source_for_Status), 29)
  			OR SHL(BYTE_TO_DWORD(cmd_for_Status), 26)
  			OR SHL(BYTE_TO_DWORD(command_error_for_Status), 23)
  			OR SHL(BOOL_TO_DWORD(StrDIp.OpcCommandsDisabled ), 21)
  			OR SHL(BOOL_TO_DWORD(StrDIp.Signaling), 16)
  			OR SHL(BOOL_TO_DWORD(StrDIp.RunOnStart ), 15)
  			OR SHL(BOOL_TO_DWORD(StrDIp.remont), 6)
  			OR SHL(BOOL_TO_DWORD(StrDIp.Check), 5)
  			OR SHL(BOOL_TO_DWORD(StrDIp.hasError), 4)
  			OR SHL(BOOL_TO_DWORD(StrDIp.SignalingTP), 3)
  			OR SHL(BOOL_TO_DWORD(StrDIp.CanRun), 2)
  			OR SHL(BOOL_TO_DWORD(StrDIp.isEnded), 1)
  			OR BOOL_TO_DWORD(StrDIp.isRunning);
END_FUNCTION_BLOCK

FUNCTION_BLOCK proc_Protection
  VAR
    fb_mvOff : fb_MvProtection;
    fb_dPmaslo_gaz_Less100 : fb_DiProtection;
    fb_Reg_vozb_off : fb_DiProtection;
    fb_Fail_chastotnii_pusk : fb_DiProtection;
    fb_Off_avar_vikluchatel : fb_DiProtection;
    fb_AOKC_SHKC : fb_DiProtection;
    fb_AO_PRU : fb_DiProtection;
    fb_AO_ot_SHU : fb_DiProtection;
    fb_Kran1_sdvig : fb_KranOpenProtection;
    fb_Kran2_sdvig : fb_KranOpenProtection;
    fb_Toporno_podshipnika_EDT_1 : fb_AiProtection;
    fb_Toy_podshipnika_EDT_2 : fb_AiProtection;
    fb_Toy_podshipnika_kol_EDT_3 : fb_AiProtection;
    fb_Toy_podshipnika_kol_EDT_4 : fb_AiProtection;
    fb_Toy_podshipnika_shest_red_EDT_5 : fb_AiProtection;
    fb_Ty_podshipnika_red_EDT_6 : fb_AiProtection;
    fb_Ty_podshipnika_nagnet_EDT_7_1 : fb_AiProtection;
    fb_Ty_podshipnika_nagnet_EDT_7_2 : fb_AiProtection;
    fb_Toy_podshipnika_svobod_konca_EDT_8_1 : fb_AiProtection;
    fb_Toy_podshipnika_svobod_konca_EDT_8_2 : fb_AiProtection;
    fb_Toy_podshipnika_rab_kol_EDT_9_1 : fb_AiProtection;
    fb_Toy_podshipnika_rab_kol_EDT_9_2 : fb_AiProtection;
    fb_Toy_podshipnika_nerab_kol_EDT_10_1 : fb_AiProtection;
    fb_Toy_podshipnika_nerab_kol_EDT_10_2 : fb_AiProtection;
    fb_Tgaza_na_vhode_H : fb_AiProtection;
    fb_Tgaza_na_vyhode_H : fb_AiProtection;
    fb_Tmasla_v_mb : fb_AiProtection;
    fb_Tmasla_v_mb_nad_ten : fb_AiProtection;
    fb_Tgorjachego_vozduha_ED_kanal_1 : fb_AiProtection;
    fb_Tgorjachego_vozduha_ED_kanal_2 : fb_AiProtection;
    fb_Tmasla_do_AVOM : fb_AiProtection;
    fb_Tmasla_posle_AVOM : fb_AiProtection;
    fb_Tmedi_statora_kanal_1 : fb_AiProtection;
    fb_Tmedi_statora_kanal_2 : fb_AiProtection;
    fb_Tmedi_statora_kanal_3 : fb_AiProtection;
    fb_Tstali_statora_kanal_1 : fb_AiProtection;
    fb_Tstali_statora_kanal_2 : fb_AiProtection;
    fb_Tstali_statora_kanal_3 : fb_AiProtection;
    fb_Tholodnogo_vozduha_ED_kanal_1 : fb_AiProtection;
    fb_Tholodnogo_vozduha_ED_kanal_2 : fb_AiProtection;
    fb_Pmaslo_sm_nizkoe : fb_AiProtection;
    fb_Pmaslo_sm_vysokoe : fb_AiProtection;
    fb_Pgaza_na_vhode_nagnetatelia : fb_AiProtection;
    fb_Pgaza_na_vyhode_nagnetatelia : fb_AiProtection;
    fb_Pmasla_posle_NU : fb_AiProtection;
    fb_Pmasla_smazki_posle_gns : fb_AiProtection;
    fb_Pimpuls_gaz : fb_AiProtection;
    fb_dPmaslo_gaz : fb_AiProtection;
    fb_dP_maslo_na_filtre : fb_AiProtection;
    fb_Os_sdvig_nagnetatelja_plus : fb_AiProtection;
    fb_Os_sdvig_nagnetatelja_minus : fb_AiProtection;
    fb_Vibro_skorost_OPED_T1 : fb_AiProtection;
    fb_Vibro_skorost_OPED_T2 : fb_AiProtection;
    fb_Vibro_skorost_OYP_kolesa_ED_T3 : fb_AiProtection;
    fb_Vibro_skorost_OP_kolesa_RH_T4 : fb_AiProtection;
    fb_Vibro_skorost_OP_shesterni_RED_T5 : fb_AiProtection;
    fb_Vibro_skorost_OP_shesterni_RED_T6 : fb_AiProtection;
    fb_Vibroperemesh_vala_N_T7 : fb_AiProtection;
    fb_Vibroperemesh_vala_N_T8 : fb_AiProtection;
    fb_Uroven_masla_v_mb : fb_AiProtection;
    fb_Tok_statora : fb_AiProtection;
    fb_Kontrol_per_220V_less187 : fb_AiProtection;
    fb_Kontrol_per_220V_high242 : fb_AiProtection;
    fb_Kontrol_post_220V_less187 : fb_AiProtection;
    fb_Kontrol_post_220V_high242 : fb_AiProtection;
  END_VAR
  VAR_EXTERNAL
    protections : ProtectionsConfig;
    ai : AiConfig;
    IM : ImConfig;
  END_VAR

  (************************************************************* DiProtection ************************************************************)
  (* МВ отключен
  fb_mvOff(sw:=IM.mv, StrDIp := protections.Pgaza_na_vyhode_nagnetatelia_GPA_STOP);*)

  (* Неисправность возбудительного устройства *)
  fb_dPmaslo_gaz_Less100(di := IM.SingleSignals.dP_maslo_gaz_Less100, StrDIp := protections.dPmaslo_gaz_less100);

  (* Сдвиг крана №2 *)
  fb_Reg_vozb_off(di:=IM.SingleSignals.Vozbud_neispravnost, StrDIp := protections.Reg_vozb_off);

  (* Сдвиг крана №2 *)
  fb_Fail_chastotnii_pusk(di:=IM.SingleSignals.Neuspesh_chastotny_pusk, StrDIp := protections.Fail_chastotnii_pusk);

  (* Сдвиг крана №2 *)
  fb_Off_avar_vikluchatel(di:=IM.SingleSignals.Avariinoe_otkluch_vikluchatelya, StrDIp := protections.Off_avar_vikluchatel);

  (* Сдвиг крана №2 *)
  fb_AOKC_SHKC(di:=IM.SingleSignals.AO_KC_ot_SHKS, StrDIp := protections.AOKC_SHKC);

  (* Сдвиг крана №2 *)
  fb_AO_PRU(di:=IM.SingleSignals.AO_GPA_ot_PRU, StrDIp := protections.AO_PRU);

  (* Сдвиг крана №2 *)
  fb_AO_ot_SHU(di:=IM.SingleSignals.AO_GPA_ot_SHU, StrDIp := protections.AO_ot_SHU);

  (* Сдвиг крана №2 *)
  fb_Kran1_sdvig(im:=IM.Kran1, StrDIp := protections.Kran1_sdvig);

  (* Сдвиг крана №2 *)
  fb_Kran2_sdvig(im:=IM.Kran2, StrDIp := protections.Kran2_sdvig);

  (************************************************************* AiProtection ************************************************************)

  (* Температура переднего опорного подшипника двигателя, т.1 *)
  fb_Toporno_podshipnika_EDT_1(ai := ai.Toporno_podshipnika_EDT_1, StrAIp := protections.Topornogo_podshipnika_EDT_1);

  (* Температура заднего опорного подшипника двигателя, т.2 *)
  fb_Toy_podshipnika_EDT_2(ai := ai.Toy_podshipnika_EDT_2, StrAIp := protections.Toy_podshipnika_EDT_2);

  (* Температура подшипника редуктора, т1 *)
  fb_Toy_podshipnika_kol_EDT_3(ai := ai.Toy_podshipnika_kol_EDT_3, StrAIp := protections.Toy_podshipnika_kol_EDT_3);

  (* Температура подшипника редуктора, т2 *)
  fb_Toy_podshipnika_kol_EDT_4(ai := ai.Toy_podshipnika_kol_EDT_4, StrAIp := protections.Toy_podshipnika_kol_EDT_4);

  (* Температура подшипника редуктора, т3 *)
  fb_Toy_podshipnika_shest_red_EDT_5(ai := ai.Toy_podshipnika_shest_red_EDT_5, StrAIp := protections.To_podshipnika_shest_red_EDT_5);

  (* Температура подшипника редуктора, т4 *)
  fb_Ty_podshipnika_red_EDT_6(ai := ai.Ty_podshipnika_red_EDT_6, StrAIp := protections.To_podshipnika_shest_red_EDT_6);

  (* Температура опорного подшипника нагнетателя, т1 *)
  fb_Ty_podshipnika_nagnet_EDT_7_1(ai := ai.Ty_podshipnika_nagnet_EDT_7_1, StrAIp := protections.To_podshipnika_N_EDT_7);

  (* Температура опорного подшипника нагнетателя, т1 *)
  fb_Ty_podshipnika_nagnet_EDT_7_2(ai := ai.Ty_podshipnika_nagnet_EDT_7_2, StrAIp := protections.To_podshipnika_N_EDT_7);

  (* Температура опорного подшипника нагнетателя, т2 *)
  fb_Toy_podshipnika_svobod_konca_EDT_8_1(ai := ai.Toy_podshipnika_svobod_konca_EDT_8_1, StrAIp := protections.To_podshipnika_svob_konca_EDT_8);

  (* Температура опорного подшипника нагнетателя, т2 *)
  fb_Toy_podshipnika_svobod_konca_EDT_8_2(ai := ai.Toy_podshipnika_svobod_konca_EDT_8_2, StrAIp := protections.To_podshipnika_svob_konca_EDT_8);

  (* Температура опорного подшипника нагнетателя, т3 *)
  fb_Toy_podshipnika_rab_kol_EDT_9_1(ai := ai.Toy_podshipnika_rab_kol_EDT_9_1, StrAIp := protections.Ty_podshipnika_rab_kol_EDT_9);

  (* Температура опорного подшипника нагнетателя, т3 *)
  fb_Toy_podshipnika_rab_kol_EDT_9_2(ai := ai.Toy_podshipnika_rab_kol_EDT_9_2, StrAIp := protections.Ty_podshipnika_rab_kol_EDT_9);

  (* Температура упорно опорного подшипника нагнетателя, т4 *)
  fb_Toy_podshipnika_nerab_kol_EDT_10_1(ai := ai.Toy_podshipnika_nerab_kol_EDT_10_1, StrAIp := protections.Typornogo_podshipnika_nerab_kolodok_HT_10);

  (* Температура упорно опорного подшипника нагнетателя, т4 *)
  fb_Toy_podshipnika_nerab_kol_EDT_10_2(ai := ai.Toy_podshipnika_nerab_kol_EDT_10_2, StrAIp := protections.Typornogo_podshipnika_nerab_kolodok_HT_10);

  (* Температура газа на выходе нагнетателя *)
  fb_Tgaza_na_vyhode_H(ai := ai.Tgaza_na_vhode_H, StrAIp := protections.Tgaza_na_vyhode_H);

  (* Температура газа на выходе нагнетателя *)
  fb_Os_sdvig_nagnetatelja_plus(ai := ai.Os_sdvig_nagnetatelja_plus, StrAIp := protections.Os_sdvig_nagnetatelja_plus);

  (* Температура газа на выходе нагнетателя *)
  fb_Os_sdvig_nagnetatelja_minus(ai := ai.Os_sdvig_nagnetatelja_minus, StrAIp := protections.Os_sdvig_nagnetatelja_minus);

  (* Температура газа на выходе нагнетателя *)
  fb_Pgaza_na_vyhode_nagnetatelia(ai := ai.Pgaza_na_vyhode_nagnetatelia, StrAIp := protections.Pgaza_na_vyhode_nagnetatelia);

  (* Температура газа на выходе нагнетателя *)
  fb_dPmaslo_gaz(ai := ai.dPmaslo_gaz, StrAIp := protections.dPmaslo_gaz);

  (* Температура газа на выходе нагнетателя *)
  fb_Pmaslo_sm_nizkoe(ai := ai.Pmaslo_sm_nizkoe, StrAIp := protections.Pmaslo_sm_nizkoe);

  (* Температура газа на выходе нагнетателя *)
  fb_Pmaslo_sm_vysokoe(ai := ai.Pmaslo_sm_vysokoe, StrAIp := protections.Pmaslo_sm_vysokoe);

  (* Температура газа на выходе нагнетателя *)
  fb_Vibro_skorost_OPED_T1(ai := ai.Vibro_skorost_OPED_T1, StrAIp := protections.Vibro_skorost_OPED_T1);

  (* Температура газа на выходе нагнетателя *)
  fb_Vibro_skorost_OPED_T2(ai := ai.Vibro_skorost_OYPED_T2, StrAIp := protections.Vibro_skorost_OPED_T2);

  (* Температура газа на выходе нагнетателя *)
  fb_Vibro_skorost_OYP_kolesa_ED_T3(ai := ai.Vibro_skorost_OYP_kolesa_ED_T3, StrAIp := protections.Vibro_skorost_OYP_kolesa_ED_T3);

  (* Температура газа на выходе нагнетателя *)
  fb_Vibro_skorost_OP_kolesa_RH_T4(ai := ai.Vibro_skorost_OP_kolesa_RH_T4, StrAIp := protections.Vibro_skorost_OP_kolesa_RH_T4);

  (* Температура газа на выходе нагнетателя *)
  fb_Vibro_skorost_OP_shesterni_RED_T5(ai := ai.Vibro_skorost_OP_shesterni_RED_T5, StrAIp := protections.Vibro_skorost_OP_shesterni_RED_T5);

  (* Температура газа на выходе нагнетателя *)
  fb_Vibro_skorost_OP_shesterni_RED_T6(ai := ai.Vibro_skorost_OP_shesterni_RED_T6, StrAIp := protections.Vibro_skorost_OP_shesterni_RED_T6);
END_FUNCTION_BLOCK

FUNCTION_BLOCK fb_Switch_Init
  VAR_INPUT
    data_Ini : BOOL;
    ISVALIDREF_statOn : BOOL;
    ISVALIDREF_statOff : BOOL;
    ISVALIDREF_cmdOn : BOOL;
    ISVALIDREF_cmdOff : BOOL;
    ISVALIDREF_inBreakCmdOn : BOOL;
    ISVALIDREF_inBreakCmdOff : BOOL;
  END_VAR
  VAR_IN_OUT
    str_Sw : struct_Switch;
  END_VAR
  VAR_OUTPUT
    Init : BOOL      := FALSE;
  END_VAR

  (*****            Функциональный блок переинициализации структуры  Switch          *****)

   Init := FALSE;

      IF data_Ini THEN                            (* Параметрам требуется переинициализация. *)
          str_Sw.ISVALIDREF_statOn                := ISVALIDREF_statOn;
          str_Sw.ISVALIDREF_statOff               := ISVALIDREF_statOff;
          str_Sw.ISVALIDREF_cmdOn                 := ISVALIDREF_cmdOn;
          str_Sw.ISVALIDREF_cmdOff                := ISVALIDREF_cmdOff;
          str_Sw.ISVALIDREF_inBreakCmdOn          := ISVALIDREF_inBreakCmdOn;
          str_Sw.ISVALIDREF_inBreakCmdOff         := ISVALIDREF_inBreakCmdOff;
          data_Ini:=FALSE;
          Init := TRUE;
      END_IF;
  IF Init THEN
          ISVALIDREF_statOn:= FALSE;
          ISVALIDREF_statOff:= FALSE;
          ISVALIDREF_cmdOn:= FALSE;
          ISVALIDREF_cmdOff:= FALSE;
          ISVALIDREF_inBreakCmdOn:= FALSE;
          ISVALIDREF_inBreakCmdOff:= FALSE;
  END_IF;
END_FUNCTION_BLOCK

FUNCTION_BLOCK fb_OilPump_Init
  VAR_INPUT
    data_Ini : BOOL;
    ISVALIDREF_statOn : BOOL;
    ISVALIDREF_statOff : BOOL;
    ISVALIDREF_cmdOn : BOOL;
    ISVALIDREF_cmdOff : BOOL;
    ISVALIDREF_inBreakCmdOn : BOOL;
    ISVALIDREF_inBreakCmdOff : BOOL;
  END_VAR
  VAR_IN_OUT
    str_Op : struct_OilPump;
  END_VAR
  VAR_OUTPUT
    Init : BOOL      := FALSE;
  END_VAR

  (*****            Функциональный блок переинициализации структуры  НУ          *****)

   Init := FALSE;

      IF data_Ini THEN                            (* Параметрам требуется переинициализация. *)
          str_Op.ISVALIDREF_statOn                := ISVALIDREF_statOn;
          str_Op.ISVALIDREF_statOff               := ISVALIDREF_statOff;
          str_Op.ISVALIDREF_cmdOn                 := ISVALIDREF_cmdOn;
          str_Op.ISVALIDREF_cmdOff                := ISVALIDREF_cmdOff;
          str_Op.ISVALIDREF_inBreakCmdOn          := ISVALIDREF_inBreakCmdOn;
          str_Op.ISVALIDREF_inBreakCmdOff         := ISVALIDREF_inBreakCmdOff;
          data_Ini:=FALSE;
          Init := TRUE;
      END_IF;

          ISVALIDREF_statOn:= FALSE;
          ISVALIDREF_statOff:= FALSE;
          ISVALIDREF_cmdOn:= FALSE;
          ISVALIDREF_cmdOff:= FALSE;
          ISVALIDREF_inBreakCmdOn:= FALSE;
          ISVALIDREF_inBreakCmdOff:= FALSE;
END_FUNCTION_BLOCK

FUNCTION_BLOCK fb_SectionSwitch_Init
  VAR_INPUT
    data_Ini : BOOL;
    ISVALIDREF_statOn : BOOL;
    ISVALIDREF_statOff : BOOL;
    ISVALIDREF_cmdOn : BOOL;
    ISVALIDREF_cmdOff : BOOL;
    ISVALIDREF_inBreakCmdOn : BOOL;
    ISVALIDREF_inBreakCmdOff : BOOL;
    ISVALIDREF_basketRolledIn : BOOL;
    ISVALIDREF_basketRolledOut : BOOL;
    ISVALIDREF_basketTest : BOOL;
  END_VAR
  VAR_IN_OUT
    str_Sw : struct_SectionSwitch;
  END_VAR
  VAR_OUTPUT
    Init : BOOL      := FALSE;
  END_VAR

  (*****            Функциональный блок переинициализации структуры  МВ          *****)

   Init := FALSE;

      IF data_Ini THEN                            (* Параметрам требуется переинициализация. *)
          str_Sw.ISVALIDREF_statOn                := ISVALIDREF_statOn;
          str_Sw.ISVALIDREF_statOff               := ISVALIDREF_statOff;
          str_Sw.ISVALIDREF_cmdOn                 := ISVALIDREF_cmdOn;
          str_Sw.ISVALIDREF_cmdOff                := ISVALIDREF_cmdOff;
          str_Sw.ISVALIDREF_inBreakCmdOn          := ISVALIDREF_inBreakCmdOn;
          str_Sw.ISVALIDREF_inBreakCmdOff         := ISVALIDREF_inBreakCmdOff;
          str_Sw.ISVALIDREF_basketRolledIn        := ISVALIDREF_basketRolledIn;
          str_Sw.ISVALIDREF_basketRolledOut       := ISVALIDREF_basketRolledOut;
          str_Sw.ISVALIDREF_basketTest            := ISVALIDREF_basketTest;
          data_Ini:=FALSE;
          Init := TRUE;
      END_IF;
  IF Init THEN
          ISVALIDREF_statOn:= FALSE;
          ISVALIDREF_statOff:= FALSE;
          ISVALIDREF_cmdOn:= FALSE;
          ISVALIDREF_cmdOff:= FALSE;
          ISVALIDREF_inBreakCmdOn:= FALSE;
          ISVALIDREF_inBreakCmdOff:= FALSE;
          ISVALIDREF_basketRolledIn:= FALSE;
          ISVALIDREF_basketRolledOut:= FALSE;
          ISVALIDREF_basketTest:= FALSE;
  END_IF;
END_FUNCTION_BLOCK

FUNCTION_BLOCK fb_DiscretParametr_Init
  VAR_INPUT
    data_Ini : BOOL;
    currentValue : UINT;
  END_VAR
  VAR_IN_OUT
    strDp : struct_DiscretParametr;
  END_VAR
  VAR_OUTPUT
    Init : BOOL      := FALSE;
  END_VAR

  (*****            Функциональный блок переинициализации дискретного параметра.          *****)

   Init := FALSE;

      IF data_Ini THEN                            (* Параметрам требуется переинициализация. *)
          strDp.currentValue       := currentValue;
          data_Ini:=FALSE;
          Init := TRUE;
      END_IF;
  IF Init THEN
  currentValue:=0;
  END_IF;
END_FUNCTION_BLOCK

FUNCTION_BLOCK fb_singleSignal_Init
  VAR_INPUT
    data_Ini : BOOL;
    inverse : BOOL;
    DelayOn : TIME;
    DelayOff : TIME;
  END_VAR
  VAR_IN_OUT
    str_SS : struct_singleSignal;
  END_VAR
  VAR_OUTPUT
    Init : BOOL      := FALSE;
  END_VAR

  (*****            Функциональный блок переинициализации структуры  singleSignal          *****)
  Init := FALSE;

      IF data_Ini THEN                            (* Параметрам требуется переинициализация. *)
          str_SS.inverse                := inverse;
          str_SS.DelayOn                := DelayOn;
          str_SS.DelayOff               := DelayOff;

          data_Ini:=FALSE;
          Init := TRUE;
      END_IF;
   IF Init THEN
          inverse := FALSE;
          DelayOn := T#0S;
          DelayOff:= T#0S;
   END_IF;
END_FUNCTION_BLOCK

FUNCTION_BLOCK fb_singleOutput_Init
  VAR_INPUT
    data_Ini : BOOL;
    inOpcCommandsDisabled : BOOL;
    wait_time : TIME;
  END_VAR
  VAR_IN_OUT
    str_SO : struct_singleOutput;
  END_VAR
  VAR_OUTPUT
    Init : BOOL      := FALSE;
  END_VAR

  (*****            Функциональный блок переинициализации структуры  singleOutput          *****)

  Init := FALSE;

      IF data_Ini THEN                            (* Параметрам требуется переинициализация. *)
          str_SO.inOpcCommandsDisabled    := inOpcCommandsDisabled;
          str_SO.wait_time                := wait_time;

           data_Ini:=FALSE;
          Init := TRUE;
      END_IF;
   IF Init THEN
          inOpcCommandsDisabled := FALSE;
          wait_time := T#0S;
     END_IF;
END_FUNCTION_BLOCK

FUNCTION_BLOCK proc_IM_Init
  VAR_INPUT
    init : BOOL;
  END_VAR
  VAR
    stKr_Ini : fb_Kran_Init;
    stSw_Ini : fb_Switch_Init;
    stOp_Ini : fb_OilPump_Init;
    stSSw_Ini : fb_SectionSwitch_Init;
    stAp_Ini : fb_AnalogParametr_Init;
    stDp_Ini : fb_DiscretParametr_Init;
    stSs_Ini : fb_singleSignal_Init;
    stSo_Ini : fb_singleOutput_Init;
    inits : UINT;
  END_VAR
  VAR_INPUT
    initiales : UINT;
  END_VAR
  VAR_EXTERNAL
    IM : ImConfig;
  END_VAR

  inits := 0; (* Флаг необходимости инициализации структур-дескрипторов *)
                                       (* Стартовая инициализация ИМ *)
  (* Кран 1 *)
  stKr_Ini(data_Ini := true, ISVALIDREF_statOn:=true, ISVALIDREF_statOff:=true,
        ISVALIDREF_cmdOn:=true, ISVALIDREF_cmdOff:=true,
        ISVALIDREF_inSo:=true, ISVALIDREF_inSz:=true,
        str_Kr := IM.Kran1);
  inits := inits + BOOL_TO_UINT(stKr_Ini.Init);

  (* Кран 2 *)
  stKr_Ini(data_Ini := true, ISVALIDREF_statOn:=true, ISVALIDREF_statOff:=true,
        ISVALIDREF_cmdOn:=true, ISVALIDREF_cmdOff:=true,
        ISVALIDREF_inSo:=true, ISVALIDREF_inSz:=true,
        str_Kr := IM.Kran2);
  inits := inits + BOOL_TO_UINT(stKr_Ini.Init);

  (* Кран 3 *)
  stKr_Ini(data_Ini := true, ISVALIDREF_statOn:=true, ISVALIDREF_statOff:=true,
        ISVALIDREF_cmdOn:=true, ISVALIDREF_cmdOff:=true,
        ISVALIDREF_inSo:=true, ISVALIDREF_inSz:=true,
        str_Kr := IM.Kran3);
  inits := inits + BOOL_TO_UINT(stKr_Ini.Init);

  (* Кран 3b *)
  stKr_Ini(data_Ini := true, ISVALIDREF_statOn:=true, ISVALIDREF_statOff:=true,
        ISVALIDREF_cmdOn:=true, ISVALIDREF_cmdOff:=true,
        ISVALIDREF_inSo:=true, ISVALIDREF_inSz:=true,
        str_Kr := IM.Kran3b);
  inits := inits + BOOL_TO_UINT(stKr_Ini.Init);

  (* Кран 4 *)
  stKr_Ini(data_Ini := true, ISVALIDREF_statOn:=true, ISVALIDREF_statOff:=true,
        ISVALIDREF_cmdOn:=true, ISVALIDREF_cmdOff:=true,
        ISVALIDREF_inSo:=true, ISVALIDREF_inSz:=true,
        str_Kr := IM.Kran4);
  inits := inits + BOOL_TO_UINT(stKr_Ini.Init);

  (* Кран 5 *)
  stKr_Ini(data_Ini := true, ISVALIDREF_statOn:=true, ISVALIDREF_statOff:=true,
        ISVALIDREF_cmdOn:=true, ISVALIDREF_cmdOff:=true,
        ISVALIDREF_inSo:=true, ISVALIDREF_inSz:=true, continueHoldCommand:=T#5S,
        str_Kr := IM.Kran5);
  inits := inits + BOOL_TO_UINT(stKr_Ini.Init);

  (* Кран 6 *)
  stKr_Ini(data_Ini := true, ISVALIDREF_statOn:=true, ISVALIDREF_statOff:=true,
        ISVALIDREF_cmdOn:=true, ISVALIDREF_cmdOff:=true,
        str_Kr := IM.Kran6);
  inits := inits + BOOL_TO_UINT(stKr_Ini.Init);

  (* НУ1 Насос уплотнения *)
  stOp_Ini(data_Ini := true, ISVALIDREF_statOn:=true, ISVALIDREF_statOff:=true,
        ISVALIDREF_cmdOn:=true, ISVALIDREF_cmdOff:=true,
        str_Op := IM.nu1);
  inits := inits + BOOL_TO_UINT(stOp_Ini.Init);

  (* НУ2 Насос уплотнения *)
  stOp_Ini(data_Ini := true, ISVALIDREF_statOn:=true, ISVALIDREF_statOff:=true,
        ISVALIDREF_cmdOn:=true, ISVALIDREF_cmdOff:=true,
        str_Op := IM.nu2);
  inits := inits + BOOL_TO_UINT(stOp_Ini.Init);

  (* ПНС Насос смазки *)
  stSw_Ini(data_Ini := true, ISVALIDREF_statOn:=true, ISVALIDREF_statOff:=true,
        ISVALIDREF_cmdOn:=true, ISVALIDREF_cmdOff:=true,
        str_Sw := IM.pns);
  inits := inits + BOOL_TO_UINT(stSw_Ini.Init);

  (* В1 АВОМ вентилятор охлаждения *)
  stSw_Ini(data_Ini := true, ISVALIDREF_statOn:=true, ISVALIDREF_statOff:=true,
        ISVALIDREF_cmdOn:=true, ISVALIDREF_cmdOff:=true,
        str_Sw := IM.v1_Avom);
  inits := inits + BOOL_TO_UINT(stSw_Ini.Init);

  (* В2 АВОМ вентилятор охлаждения *)
  stSw_Ini(data_Ini := true, ISVALIDREF_statOn:=true, ISVALIDREF_statOff:=true,
        ISVALIDREF_cmdOn:=true, ISVALIDREF_cmdOff:=true,
        str_Sw := IM.v2_Avom);
  inits := inits + BOOL_TO_UINT(stSw_Ini.Init);

  (* В3 АВОМ вентилятор охлаждения *)
  stSw_Ini(data_Ini := true, ISVALIDREF_statOn:=true, ISVALIDREF_statOff:=true,
        ISVALIDREF_cmdOn:=true, ISVALIDREF_cmdOff:=true,
        str_Sw := IM.v3_Avom);
  inits := inits + BOOL_TO_UINT(stSw_Ini.Init);

  (* В4 АВОМ вентилятор охлаждения *)
  stSw_Ini(data_Ini := true, ISVALIDREF_statOn:=true, ISVALIDREF_statOff:=true,
        ISVALIDREF_cmdOn:=true, ISVALIDREF_cmdOff:=true,
        str_Sw := IM.v4_Avom);
  inits := inits + BOOL_TO_UINT(stSw_Ini.Init);

  (* МВ масляный выключатель *)
  stSSw_Ini(data_Ini := true, ISVALIDREF_statOn:=true, ISVALIDREF_statOff:=true,
        ISVALIDREF_cmdOn:=true, ISVALIDREF_cmdOff:=true,
        ISVALIDREF_basketRolledIn:=true, ISVALIDREF_basketRolledout:=true,
        str_Sw := IM.mv);
  inits := inits + BOOL_TO_UINT(stSSw_Ini.Init);

  (* В4 АВОМ вентилятор охлаждения *)
  stSw_Ini(data_Ini := true, ISVALIDREF_statOn:=true, ISVALIDREF_statOff:=true,
        ISVALIDREF_cmdOn:=true, ISVALIDREF_cmdOff:=true,
        str_Sw := IM.KaloriferAVOM);
  inits := inits + BOOL_TO_UINT(stSw_Ini.Init);

  (* В4 АВОМ вентилятор охлаждения *)
  stSw_Ini(data_Ini := true, ISVALIDREF_statOn:=true, ISVALIDREF_statOff:=true,
        ISVALIDREF_cmdOn:=true, ISVALIDREF_cmdOff:=true,
        str_Sw := IM.CMN);
  inits := inits + BOOL_TO_UINT(stSw_Ini.Init);

  (* В4 АВОМ вентилятор охлаждения *)
  stSw_Ini(data_Ini := true, ISVALIDREF_statOn:=true, ISVALIDREF_statOff:=true,
        ISVALIDREF_cmdOn:=true, ISVALIDREF_cmdOff:=true,
        str_Sw := IM.TEN_kollectora);
  inits := inits + BOOL_TO_UINT(stSw_Ini.Init);

  (* В4 АВОМ вентилятор охлаждения *)
  stSw_Ini(data_Ini := true, ISVALIDREF_statOn:=true, ISVALIDREF_statOff:=true,
        ISVALIDREF_cmdOn:=true, ISVALIDREF_cmdOff:=true,
        str_Sw := IM.TEN_MB);
  inits := inits + BOOL_TO_UINT(stSw_Ini.Init);

                                       (* Стартовая инициализация singleSignal *)
      (* Перепад давления «газ-газ» на кране 1 ≤1 кгс/см² *)
  stSs_Ini(data_Ini := true, inverse:=FALSE, (*DelayOn:=T#0S, DelayOff:=T#0S,*) str_SS := IM.SingleSignals.dP_maslo_gaz_Less100);
  inits := inits + BOOL_TO_UINT(stSs_Ini.Init);

   (* Осевой сдвиг ротора вправо ≥3,7 кгс/см² *)
  stSs_Ini(data_Ini := true, inverse:=FALSE, (*DelayOn:=T#0S, DelayOff:=T#0S,*) str_SS := IM.SingleSignals.dp_kran1_Less100);
  inits := inits + BOOL_TO_UINT(stSs_Ini.Init);

      (* Пробой вентиля *)
  stSs_Ini(data_Ini := true, inverse:=TRUE, (*DelayOn:=T#0S, DelayOff:=T#0S,*) str_SS := IM.SingleSignals.Vozbud_neispr_tsepey_upr_AVR_pit);
  inits := inits + BOOL_TO_UINT(stSs_Ini.Init);

      (* Работа схемы ресинхронизации *)
  stSs_Ini(data_Ini := true, inverse:=FALSE, (*DelayOn:=T#0S, DelayOff:=T#0S,*) str_SS := IM.SingleSignals.Vozbud_gotovnost);
  inits := inits + BOOL_TO_UINT(stSs_Ini.Init);

      (* Контроль состояния возбудительного устройства  *)
  stSs_Ini(data_Ini := true, inverse:=FALSE, (*DelayOn:=T#0S, DelayOff:=T#0S,*) str_SS := IM.SingleSignals.Vozbud_neispravnost);
  inits := inits + BOOL_TO_UINT(stSs_Ini.Init);

      (* Неисправность форсировки воз-буждения  *)
  stSs_Ini(data_Ini := true, inverse:=FALSE, (*DelayOn:=T#0S, DelayOff:=T#0S,*) str_SS := IM.SingleSignals.SHAVR1_v_rabote);
  inits := inits + BOOL_TO_UINT(stSs_Ini.Init);

    (* Неисправность возбудительного устройства  *)
  stSs_Ini(data_Ini := true, inverse:=FALSE, (*DelayOn:=T#0S, DelayOff:=T#0S,*) str_SS := IM.SingleSignals.SHAVR2_v_rabote);
  inits := inits + BOOL_TO_UINT(stSs_Ini.Init);

    (* Готовность включения БЭО по отказу контроллера  *)
  stSs_Ini(data_Ini := true, inverse:=FALSE, (*DelayOn:=T#0S, DelayOff:=T#0S,*) str_SS := IM.SingleSignals.Avariinoe_otkluch_vikluchatelya);
  inits := inits + BOOL_TO_UINT(stSs_Ini.Init);

    (* Срабатывание БЭАО  *)
  stSs_Ini(data_Ini := true, inverse:=FALSE, (*DelayOn:=T#0S, DelayOff:=T#0S,*) str_SS := IM.SingleSignals.Assinhronnii_hod_peregruzka);
  inits := inits + BOOL_TO_UINT(stSs_Ini.Init);

    (* Выключатель основного ввода питания QF1  в положении включен   *)
  stSs_Ini(data_Ini := true, inverse:=TRUE, (*DelayOn:=T#0S, DelayOff:=T#0S,*) str_SS := IM.SingleSignals.QF1_on);
  inits := inits + BOOL_TO_UINT(stSs_Ini.Init);

    (* Выключатель резервного ввода питания QF2  в положении включен   *)
  stSs_Ini(data_Ini := true, inverse:=TRUE, (*DelayOn:=T#0S, DelayOff:=T#0S,*) str_SS := IM.SingleSignals.QF2_on);
  inits := inits + BOOL_TO_UINT(stSs_Ini.Init);

    (* Выключатель питания кранов:  QF23 110 В в положении включен   *)
  stSs_Ini(data_Ini := true, inverse:=TRUE, (*DelayOn:=T#0S, DelayOff:=T#0S,*) str_SS := IM.SingleSignals.QF23_on);
  inits := inits + BOOL_TO_UINT(stSs_Ini.Init);

    (* Выключатели группы 1: QF4, QF5 в положении включен   *)
  stSs_Ini(data_Ini := true, inverse:=TRUE, (*DelayOn:=T#0S, DelayOff:=T#0S,*) str_SS := IM.SingleSignals.QF4_QF5_on);
  inits := inits + BOOL_TO_UINT(stSs_Ini.Init);

    (* Выключатели группы 2: QF6, QF7 в положении включен   *)
  stSs_Ini(data_Ini := true, inverse:=TRUE, (*DelayOn:=T#0S, DelayOff:=T#0S,*) str_SS := IM.SingleSignals.QF6_QF7_on);
  inits := inits + BOOL_TO_UINT(stSs_Ini.Init);

    (* Выключатели группы 3: QF8, QF9 в положении включен   *)
  stSs_Ini(data_Ini := true, inverse:=TRUE, (*DelayOn:=T#0S, DelayOff:=T#0S,*) str_SS := IM.SingleSignals.QF8_QF9_on);
  inits := inits + BOOL_TO_UINT(stSs_Ini.Init);

    (* Выключатели группы 4: QF10, QF11 в положении включен   *)
  stSs_Ini(data_Ini := true, inverse:=TRUE, (*DelayOn:=T#0S, DelayOff:=T#0S,*) str_SS := IM.SingleSignals.QF10_QF11_on);
  inits := inits + BOOL_TO_UINT(stSs_Ini.Init);

    (* Выключатели группы 5: QF12, QF13 в положении включен   *)
  stSs_Ini(data_Ini := true, inverse:=TRUE, (*DelayOn:=T#0S, DelayOff:=T#0S,*) str_SS := IM.SingleSignals.QF12_QF13_on);
  inits := inits + BOOL_TO_UINT(stSs_Ini.Init);

    (* Выключатели группы 6: QF14, QF15 в положении включен   *)
  stSs_Ini(data_Ini := true, inverse:=TRUE, (*DelayOn:=T#0S, DelayOff:=T#0S,*) str_SS := IM.SingleSignals.QF14_QF15_on);
  inits := inits + BOOL_TO_UINT(stSs_Ini.Init);

    (* Выключатели группы : QF22 в положении включен   *)
  stSs_Ini(data_Ini := true, inverse:=TRUE, (*DelayOn:=T#0S, DelayOff:=T#0S,*) str_SS := IM.SingleSignals.QF22_on);
  inits := inits + BOOL_TO_UINT(stSs_Ini.Init);

    (* Неисправность источников питания группы 1: G1, G2 (=24 В)   *)
  stSs_Ini(data_Ini := true, inverse:=TRUE, (*DelayOn:=T#0S, DelayOff:=T#0S,*) str_SS := IM.SingleSignals.NS_G1_G2);
  inits := inits + BOOL_TO_UINT(stSs_Ini.Init);

    (* Неисправность источников питания группы 2: G3, G4 (=24 В)   *)
  stSs_Ini(data_Ini := true, inverse:=TRUE, (*DelayOn:=T#0S, DelayOff:=T#0S,*) str_SS := IM.SingleSignals.NS_G3_G4);
  inits := inits + BOOL_TO_UINT(stSs_Ini.Init);

    (* Неисправность источников питания внутренних ПТС: G15, G16 (=24 В)   *)
  stSs_Ini(data_Ini := true, inverse:=TRUE, (*DelayOn:=T#0S, DelayOff:=T#0S,*) str_SS := IM.SingleSignals.NS_G15_G16);
  inits := inits + BOOL_TO_UINT(stSs_Ini.Init);

    (* Неисправность источника питания аналоговых сигналов: G17 (=24 В)   *)
  stSs_Ini(data_Ini := true, inverse:=TRUE, (*DelayOn:=T#0S, DelayOff:=T#0S,*) str_SS := IM.SingleSignals.NS_G17);
  inits := inits + BOOL_TO_UINT(stSs_Ini.Init);

    (* Неисправность источников питания группы 3: G5, G6 (=24 В)   *)
  stSs_Ini(data_Ini := true, inverse:=TRUE, (*DelayOn:=T#0S, DelayOff:=T#0S,*) str_SS := IM.SingleSignals.NS_G5_G6);
  inits := inits + BOOL_TO_UINT(stSs_Ini.Init);

    (* Неисправность источников питания группы 4: G7, G8 (=24 В)   *)
  stSs_Ini(data_Ini := true, inverse:=TRUE, (*DelayOn:=T#0S, DelayOff:=T#0S,*) str_SS := IM.SingleSignals.NS_G7_G8);
  inits := inits + BOOL_TO_UINT(stSs_Ini.Init);

    (* Неисправность источников питания внешних цепей: G18, G19 (=24 В)   *)
  stSs_Ini(data_Ini := true, inverse:=TRUE, (*DelayOn:=T#0S, DelayOff:=T#0S,*) str_SS := IM.SingleSignals.NS_G18_G19);
  inits := inits + BOOL_TO_UINT(stSs_Ini.Init);

    (* Неисправность источников питания группы 5: G9, G10, G11, G12 (=110 В)   *)
  stSs_Ini(data_Ini := true, inverse:=TRUE, (*DelayOn:=T#0S, DelayOff:=T#0S,*) str_SS := IM.SingleSignals.NS_G10_G11);
  inits := inits + BOOL_TO_UINT(stSs_Ini.Init);

    (* Неисправность источников питания G13, G14 (=24 В)   *)
  stSs_Ini(data_Ini := true, inverse:=TRUE, (*DelayOn:=T#0S, DelayOff:=T#0S,*) str_SS := IM.SingleSignals.NS_G13_G14);
  inits := inits + BOOL_TO_UINT(stSs_Ini.Init);

      (* Неисправность источников питания G13, G14 (=24 В)   *)
  stSs_Ini(data_Ini := true, inverse:=TRUE, (*DelayOn:=T#0S, DelayOff:=T#0S,*) str_SS := IM.SingleSignals.Uroven_masla_akkum);
  inits := inits + BOOL_TO_UINT(stSs_Ini.Init);

    (* Неисправность источников питания G13, G14 (=24 В)   *)
  stSs_Ini(data_Ini := true, inverse:=TRUE, (*DelayOn:=T#0S, DelayOff:=T#0S,*) str_SS := IM.SingleSignals.BEAO_srabotal);
  inits := inits + BOOL_TO_UINT(stSs_Ini.Init);

    (* Неисправность источников питания G13, G14 (=24 В)   *)
  stSs_Ini(data_Ini := true, inverse:=TRUE, (*DelayOn:=T#0S, DelayOff:=T#0S,*) str_SS := IM.SingleSignals.Chastotny_pusk);
  inits := inits + BOOL_TO_UINT(stSs_Ini.Init);

    (* Неисправность источников питания G13, G14 (=24 В)   *)
  stSs_Ini(data_Ini := true, inverse:=TRUE, (*DelayOn:=T#0S, DelayOff:=T#0S,*) str_SS := IM.SingleSignals.Neuspesh_chastotny_pusk);
  inits := inits + BOOL_TO_UINT(stSs_Ini.Init);

    (* Неисправность источников питания G13, G14 (=24 В)   *)
  stSs_Ini(data_Ini := true, inverse:=TRUE, (*DelayOn:=T#0S, DelayOff:=T#0S,*) str_SS := IM.SingleSignals.Rezhim_ruchnogo_regulirovaniya);
  inits := inits + BOOL_TO_UINT(stSs_Ini.Init);

    (* Неисправность источников питания G13, G14 (=24 В)   *)
  stSs_Ini(data_Ini := true, inverse:=TRUE, (*DelayOn:=T#0S, DelayOff:=T#0S,*) str_SS := IM.SingleSignals.SHU_v_GPA_vkluch);
  inits := inits + BOOL_TO_UINT(stSs_Ini.Init);

    (* Неисправность источников питания G13, G14 (=24 В)   *)
  stSs_Ini(data_Ini := true, inverse:=TRUE, (*DelayOn:=T#0S, DelayOff:=T#0S,*) str_SS := IM.SingleSignals.SHP_v_GPA_vkluch);
  inits := inits + BOOL_TO_UINT(stSs_Ini.Init);

  (* Отключение МВ1 от КНА   *)
  stSs_Ini(data_Ini := true, inverse:=TRUE, (*wait_time:=T#0S,*) str_SS := IM.SingleSignals.NKU1_GPA_on);
  inits := inits + BOOL_TO_UINT(stSs_Ini.Init);

  (* Отключение МВ1 от КНА   *)
  stSs_Ini(data_Ini := true, inverse:=TRUE, (*wait_time:=T#0S,*) str_SS := IM.SingleSignals.NKU2_GPA_on);
  inits := inits + BOOL_TO_UINT(stSs_Ini.Init);

  (* Отключение МВ1 от КНА   *)
  stSs_Ini(data_Ini := true, inverse:=TRUE, (*wait_time:=T#0S,*) str_SS := IM.SingleSignals.AO_KC_ot_SHKS);
  inits := inits + BOOL_TO_UINT(stSs_Ini.Init);

  (* Отключение МВ1 от КНА   *)
  stSs_Ini(data_Ini := true, inverse:=TRUE, (*wait_time:=T#0S,*) str_SS := IM.SingleSignals.AO_GPA_ot_SHU);
  inits := inits + BOOL_TO_UINT(stSs_Ini.Init);

  (* Отключение МВ1 от КНА   *)
  stSs_Ini(data_Ini := true, inverse:=TRUE, (*wait_time:=T#0S,*) str_SS := IM.SingleSignals.Razreshenie_zagruzki_dvig);
  inits := inits + BOOL_TO_UINT(stSs_Ini.Init);

  (* Отключение МВ1 от КНА   *)
  stSs_Ini(data_Ini := true, inverse:=TRUE, (*wait_time:=T#0S,*) str_SS := IM.SingleSignals.Osnovnoy_regul_off);
  inits := inits + BOOL_TO_UINT(stSs_Ini.Init);

  (* Отключение МВ1 от КНА   *)
  stSs_Ini(data_Ini := true, inverse:=TRUE, (*wait_time:=T#0S,*) str_SS := IM.SingleSignals.Voltage_sekcii_norm);
  inits := inits + BOOL_TO_UINT(stSs_Ini.Init);

  (* Отключение МВ1 от КНА   *)
  stSs_Ini(data_Ini := true, inverse:=TRUE, (*wait_time:=T#0S,*) str_SS := IM.SingleSignals.Reactorny_pusk);
  inits := inits + BOOL_TO_UINT(stSs_Ini.Init);

  (* Отключение МВ1 от КНА   *)
  stSs_Ini(data_Ini := true, inverse:=TRUE, (*wait_time:=T#0S,*) str_SS := IM.SingleSignals.NO_GPA_ot_SHU);
  inits := inits + BOOL_TO_UINT(stSs_Ini.Init);

  (* Отключение МВ1 от КНА   *)
  stSs_Ini(data_Ini := true, inverse:=TRUE, (*wait_time:=T#0S,*) str_SS := IM.SingleSignals.AO_GPA_ot_PRU);
  inits := inits + BOOL_TO_UINT(stSs_Ini.Init);

  (* Отключение МВ1 от КНА   *)
  stSs_Ini(data_Ini := true, inverse:=TRUE, (*wait_time:=T#0S,*) str_SS := IM.SingleSignals.Nalichie_BP1);
  inits := inits + BOOL_TO_UINT(stSs_Ini.Init);

  (* Отключение МВ1 от КНА   *)
  stSs_Ini(data_Ini := true, inverse:=TRUE, (*wait_time:=T#0S,*) str_SS := IM.SingleSignals.Nalichie_BP2);
  inits := inits + BOOL_TO_UINT(stSs_Ini.Init);

  (* Отключение МВ1 от КНА   *)
  stSs_Ini(data_Ini := true, inverse:=TRUE, (*wait_time:=T#0S,*) str_SS := IM.SingleSignals.Nalichie_BP3);
  inits := inits + BOOL_TO_UINT(stSs_Ini.Init);

  (* Отключение МВ1 от КНА   *)
  stSs_Ini(data_Ini := true, inverse:=TRUE, (*wait_time:=T#0S,*) str_SS := IM.SingleSignals.Nalichie_BP4);
  inits := inits + BOOL_TO_UINT(stSs_Ini.Init);

  (* Отключение МВ1 от КНА   *)
  stSs_Ini(data_Ini := true, inverse:=TRUE, (*wait_time:=T#0S,*) str_SS := IM.SingleSignals.Nalichie_BP5);
  inits := inits + BOOL_TO_UINT(stSs_Ini.Init);

  (* Отключение МВ1 от КНА   *)
  stSs_Ini(data_Ini := true, inverse:=TRUE, (*wait_time:=T#0S,*) str_SS := IM.SingleSignals.Nalichie_BP6);
  inits := inits + BOOL_TO_UINT(stSs_Ini.Init);

  (* Отключение МВ1 от КНА   *)
  stSs_Ini(data_Ini := true, inverse:=TRUE, (*wait_time:=T#0S,*) str_SS := IM.SingleSignals.Nalichie_BP7_BP8);
  inits := inits + BOOL_TO_UINT(stSs_Ini.Init);

  (* Отключение МВ1 от КНА   *)
  stSs_Ini(data_Ini := true, inverse:=TRUE, (*wait_time:=T#0S,*) str_SS := IM.SingleSignals.Nalichie_BP9_BP10);
  inits := inits + BOOL_TO_UINT(stSs_Ini.Init);

  (* Отключение МВ1 от КНА   *)
  stSs_Ini(data_Ini := true, inverse:=TRUE, (*wait_time:=T#0S,*) str_SS := IM.SingleSignals.Nalichie_cepei_upravlen_mv);
  inits := inits + BOOL_TO_UINT(stSs_Ini.Init);

  (* Отключение МВ1 от КНА   *)
  stSs_Ini(data_Ini := true, inverse:=TRUE, (*wait_time:=T#0S,*) str_SS := IM.SingleSignals.Nalichie_220BEAO);
  inits := inits + BOOL_TO_UINT(stSs_Ini.Init);

  (* Отключение МВ1 от КНА   *)
  stSs_Ini(data_Ini := true, inverse:=TRUE, (*wait_time:=T#0S,*) str_SS := IM.SingleSignals.Nalichie_per_220_na_vhode);
  inits := inits + BOOL_TO_UINT(stSs_Ini.Init);

  (* Отключение МВ1 от КНА   *)
  stSs_Ini(data_Ini := true, inverse:=TRUE, (*wait_time:=T#0S,*) str_SS := IM.SingleSignals.Nalichie_post_220_na_vhode);
  inits := inits + BOOL_TO_UINT(stSs_Ini.Init);

  (* Отключение МВ1 от КНА   *)
  stSs_Ini(data_Ini := true, inverse:=TRUE, (*wait_time:=T#0S,*) str_SS := IM.SingleSignals.Nalichie_BP11);
  inits := inits + BOOL_TO_UINT(stSs_Ini.Init);

  (* Отключение МВ1 от КНА   *)
  stSs_Ini(data_Ini := true, inverse:=TRUE, (*wait_time:=T#0S,*) str_SS := IM.SingleSignals.Nalichie_BP12);
  inits := inits + BOOL_TO_UINT(stSs_Ini.Init);

  (* Отключение МВ1 от КНА   *)
  stSs_Ini(data_Ini := true, inverse:=TRUE, (*wait_time:=T#0S,*) str_SS := IM.SingleSignals.Dver_SHU_pered_otkrita);
  inits := inits + BOOL_TO_UINT(stSs_Ini.Init);

  (* Отключение МВ1 от КНА   *)
  stSs_Ini(data_Ini := true, inverse:=TRUE, (*wait_time:=T#0S,*) str_SS := IM.SingleSignals.Dver_SHU_zad_otkrita);
  inits := inits + BOOL_TO_UINT(stSs_Ini.Init);

  (* Отключение МВ1 от КНА   *)
  stSs_Ini(data_Ini := true, inverse:=TRUE, (*wait_time:=T#0S,*) str_SS := IM.SingleSignals.EO_GPA_ot_knopki_SHU);
  inits := inits + BOOL_TO_UINT(stSs_Ini.Init);

  (* Отключение МВ1 от КНА   *)
  stSs_Ini(data_Ini := true, inverse:=TRUE, (*wait_time:=T#0S,*) str_SS := IM.SingleSignals.EO_EGPA_ot_PRY);
  inits := inits + BOOL_TO_UINT(stSs_Ini.Init);

  (* Отключение МВ1 от КНА   *)
  stSs_Ini(data_Ini := true, inverse:=TRUE, (*wait_time:=T#0S,*) str_SS := IM.SingleSignals.Synchroniz_rezhima_K1);
  inits := inits + BOOL_TO_UINT(stSs_Ini.Init);

                                       (* Стартовая инициализация singleOutput *)
  (* Идикация НО (подсветка кнопки на шкафу)   *)
  stSo_Ini(data_Ini := true, inOpcCommandsDisabled:=TRUE, (*wait_time:=T#0S,*) str_SO := IM.SingleOutputs.Rabota_EGPA);
  inits := inits + BOOL_TO_UINT(stSo_Ini.Init);

  (* Взвод включения БЭАО по неисправности ПТС   *)
  stSo_Ini(data_Ini := true, inOpcCommandsDisabled:=TRUE, wait_time:=T#0S, str_SO := IM.SingleOutputs.Neispr_EGPA);
  inits := inits + BOOL_TO_UINT(stSo_Ini.Init);

  (* Авария ЭГПА в КЦ   *)
  stSo_Ini(data_Ini := true, inOpcCommandsDisabled:=TRUE, (*wait_time:=T#0S,*) str_SO := IM.SingleOutputs.Avary_EGPA);
  inits := inits + BOOL_TO_UINT(stSo_Ini.Init);

  (* Авария ЭГПА в КЦ   *)
  stSo_Ini(data_Ini := true, inOpcCommandsDisabled:=TRUE, (*wait_time:=T#0S,*) str_SO := IM.SingleOutputs.U_lamp_SHU);
  inits := inits + BOOL_TO_UINT(stSo_Ini.Init);

  (* Индикация ПС Фонарь   *)
  stSo_Ini(data_Ini := true, inOpcCommandsDisabled:=TRUE, (*wait_time:=T#0S,*) str_SO := IM.SingleOutputs.AO_knopka_ind);
  inits := inits + BOOL_TO_UINT(stSo_Ini.Init);

  (* Индикация АС Фонарь   *)
  stSo_Ini(data_Ini := true, inOpcCommandsDisabled:=TRUE, (*wait_time:=T#0S,*) str_SO := IM.SingleOutputs.Pusk_SHUP);
  inits := inits + BOOL_TO_UINT(stSo_Ini.Init);

  (* Отключение МВ1 от КНА   *)
  stSo_Ini(data_Ini := true, inOpcCommandsDisabled:=TRUE, (*wait_time:=T#0S,*) str_SO := IM.SingleOutputs.Stop_SHUP);
  inits := inits + BOOL_TO_UINT(stSo_Ini.Init);

  (* Отключение МВ1 от КНА   *)
  stSo_Ini(data_Ini := true, inOpcCommandsDisabled:=TRUE, (*wait_time:=T#0S,*) str_SO := IM.SingleOutputs.NO_fonar);
  inits := inits + BOOL_TO_UINT(stSo_Ini.Init);

  (* Отключение МВ1 от КНА   *)
  stSo_Ini(data_Ini := true, inOpcCommandsDisabled:=TRUE, (*wait_time:=T#0S,*) str_SO := IM.SingleOutputs.PC_fonar);
  inits := inits + BOOL_TO_UINT(stSo_Ini.Init);

  (* Отключение МВ1 от КНА   *)
  stSo_Ini(data_Ini := true, inOpcCommandsDisabled:=TRUE, (*wait_time:=T#0S,*) str_SO := IM.SingleOutputs.AC_fonar);
  inits := inits + BOOL_TO_UINT(stSo_Ini.Init);

  (* Отключение МВ1 от КНА   *)
  stSo_Ini(data_Ini := true, inOpcCommandsDisabled:=TRUE, (*wait_time:=T#0S,*) str_SO := IM.SingleOutputs.Kr1_smazka);
  inits := inits + BOOL_TO_UINT(stSo_Ini.Init);

  (* Отключение МВ1 от КНА   *)
  stSo_Ini(data_Ini := true, inOpcCommandsDisabled:=TRUE, (*wait_time:=T#0S,*) str_SO := IM.SingleOutputs.Kr2_smazka);
  inits := inits + BOOL_TO_UINT(stSo_Ini.Init);

  (* Отключение МВ1 от КНА   *)
  stSo_Ini(data_Ini := true, inOpcCommandsDisabled:=TRUE, (*wait_time:=T#0S,*) str_SO := IM.SingleOutputs.Kr4_open_from_alg);
  inits := inits + BOOL_TO_UINT(stSo_Ini.Init);

  (* Отключение МВ1 от КНА   *)
  stSo_Ini(data_Ini := true, inOpcCommandsDisabled:=TRUE, (*wait_time:=T#0S,*) str_SO := IM.SingleOutputs.Synch_rej_K1);
  inits := inits + BOOL_TO_UINT(stSo_Ini.Init);
  initiales := 0;

  IF init THEN initiales := inits; END_IF;
END_FUNCTION_BLOCK

FUNCTION_BLOCK fb_OilPump
  VAR_INPUT
    statOn : BOOL;
    statOff : BOOL;
    statOn_reliability : BOOL;
    statOff_reliability : BOOL;
  END_VAR
  VAR_IN_OUT
    StrSw : struct_OilPump;
  END_VAR
  VAR_INPUT
    inNs : TYPE_ReliableBit;
    inAccident : TYPE_ReliableBit;
    inLocal : TYPE_ReliableBit;
    inDistance : TYPE_ReliableBit;
    inBreakCmdOn : TYPE_ReliableBit;
    inBreakCmdOff : TYPE_ReliableBit;
  END_VAR
  VAR
    onInit : BOOL      := FALSE;
    _statOn : BOOL;
    _statOff : BOOL;
    getSdvig : BOOL;
    lastOnStatus : BYTE;
    cmd : BYTE;
    source : BYTE;
    lastCmd : BYTE;
    source_for_Status : BYTE;
    cmd_for_Status : BYTE;
    command_error_for_Status : BYTE;
    _sunpackerCommand : fb_sunpackerCommand;
    _statusDualInput : TYPE_statusDualInput;
    _commandDualInput : TYPE_commandDualInput;
    _commandErrorTimer : BOOL;
    resetErrorTimer : BOOL;
    _changWithoutCommand : BOOL;
    errorCMDTimer : TON;
    sdvigReset : TON;
    _errorReset : TON;
    outputsSets : TOF;
  END_VAR
  VAR_IN_OUT
    cmdOn : BOOL;
    cmdOff : BOOL;
  END_VAR

  IF NOT onInit THEN
  IF StrSw.ISVALIDREF_cmdOn XOR StrSw.ISVALIDREF_cmdOff THEN
  	IF 	StrSw.ISVALIDREF_cmdOn THEN
  		lastCmd:= 2; (*baseCmdOff*)
  	ELSE
  		lastCmd:= 1; (*baseCmdOn*)
  	END_IF;
  END_IF;
  onInit:=TRUE;
  END_IF;

  (* ---- Если управление с ВУ заблокировано, то в ИМ передаем команду из алгоритма ---- *)
  IF StrSw.inOpcCommandsDisabled THEN
  	StrSw.inCommand := StrSw.inCommand_Alg;
  ELSE (* иначе передаем команду с АРМа*)
  	StrSw.inCommand := StrSw.inCommand_ARM;
  END_IF;

  (* ---- Формирование состояния механизма ---- *)

  IF (StrSw.ISVALIDREF_statOn) OR (StrSw.ISVALIDREF_statOff) THEN
  	IF (StrSw.ISVALIDREF_statOn) AND (StrSw.ISVALIDREF_statOff) THEN
  	StrSw.reliability:= statOn_reliability AND statOff_reliability;
  		_statOn  := statOn;
  		_statOff := statOff;
  	ELSIF (StrSw.ISVALIDREF_statOn) THEN
                       StrSw.reliability:= statOn_reliability;
  		_statOn  := statOn;
  		_statOff := NOT statOn;
  	ELSIF (StrSw.ISVALIDREF_statOff) THEN
  		 StrSw.reliability:= statOff_reliability;
  		_statOn  := NOT statOff;
  		_statOff :=statOff;
  	END_IF;
